// TIA Portal V20 export
FUNCTION "CollectAlarms" : Void   // FC66, LAD
TITLE = U1Em6_StackTable
// stored: Namespace Unit1.Em6, SetENOAutomatically false
   VAR_INPUT
      resetAlarms : Bool;
      disableAlarms : Bool;
   END_VAR
   VAR_OUTPUT
      commandsToUnit : "LUC_typeStateCommands";   // Feedback to the unit
   END_VAR
   VAR CONSTANT
      DelayTime : Time := T#300ms;
      NoDelayTime : Time;
      FALSE : Bool := FALSE;
      TRUE : Bool := TRUE;
   END_VAR
BEGIN

REGION Network 1: Reset Alarms
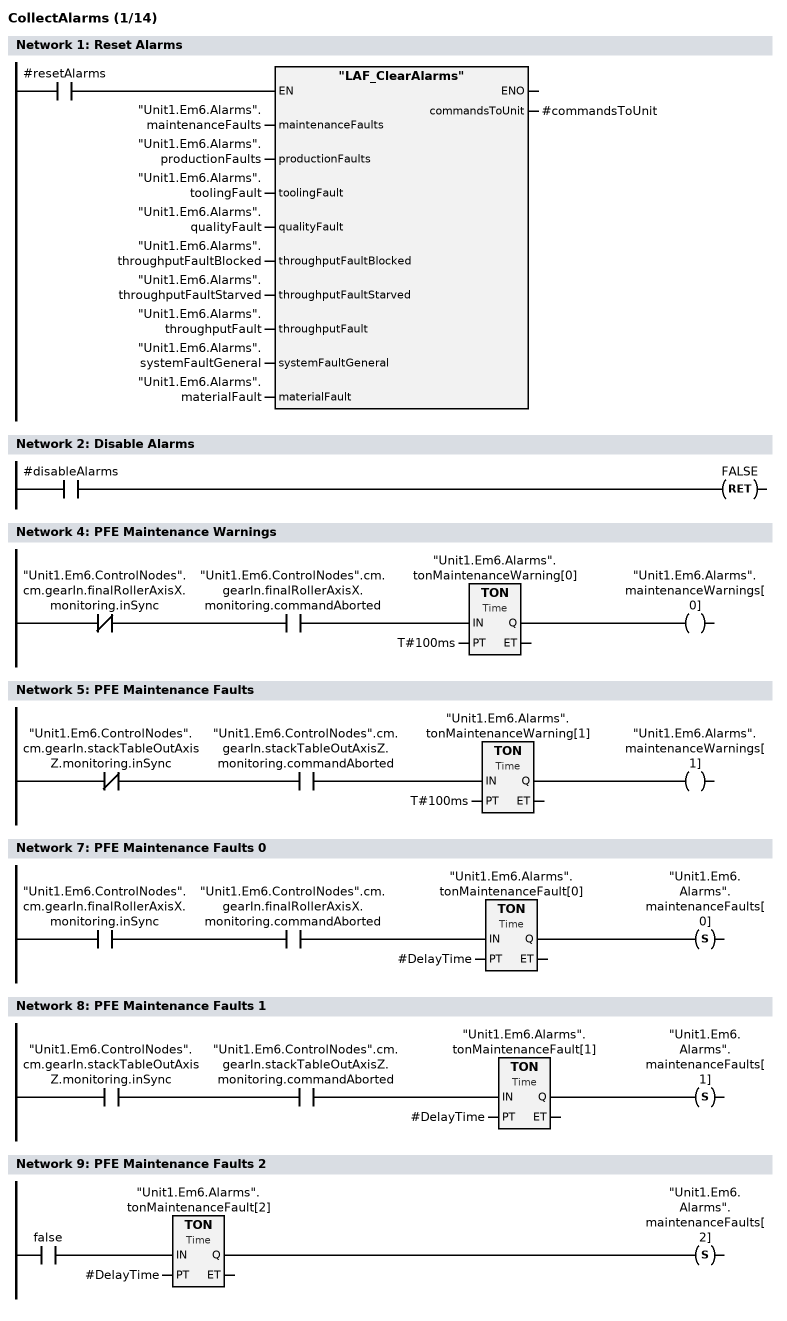
   RUNG wire#powerrail
      Contact( #resetAlarms )
      "LAF_ClearAlarms"(maintenanceFaults := "Unit1.Em6.Alarms".maintenanceFaults, productionFaults := "Unit1.Em6.Alarms".productionFaults, toolingFault := "Unit1.Em6.Alarms".toolingFault, qualityFault := "Unit1.Em6.Alarms".qualityFault, throughputFaultBlocked := "Unit1.Em6.Alarms".throughputFaultBlocked, throughputFaultStarved := "Unit1.Em6.Alarms".throughputFaultStarved, throughputFault := "Unit1.Em6.Alarms".throughputFault, systemFaultGeneral := "Unit1.Em6.Alarms".systemFaultGeneral, materialFault := "Unit1.Em6.Alarms".materialFault, commandsToUnit => #commandsToUnit)
   END_RUNG
   // the same network as SCL:
   IF #resetAlarms THEN
       "LAF_ClearAlarms"(maintenanceFaults := "Unit1.Em6.Alarms".maintenanceFaults,
                         productionFaults := "Unit1.Em6.Alarms".productionFaults,
                         toolingFault := "Unit1.Em6.Alarms".toolingFault,
                         qualityFault := "Unit1.Em6.Alarms".qualityFault,
                         throughputFaultBlocked := "Unit1.Em6.Alarms".throughputFaultBlocked,
                         throughputFaultStarved := "Unit1.Em6.Alarms".throughputFaultStarved,
                         throughputFault := "Unit1.Em6.Alarms".throughputFault,
                         systemFaultGeneral := "Unit1.Em6.Alarms".systemFaultGeneral,
                         materialFault := "Unit1.Em6.Alarms".materialFault,
                         commandsToUnit => #commandsToUnit);
   END_IF;
END_REGION

REGION Network 2: Disable Alarms
   RUNG wire#powerrail
      Contact( #disableAlarms )
      ReturnCoil( FALSE )
   END_RUNG
   // the same network as SCL:
   IF #disableAlarms THEN
       ENO := FALSE;
       RETURN;
   END_IF;
END_REGION

REGION Network 3: *************** Fault ************************
END_REGION

REGION Network 4: PFE Maintenance Warnings
   RUNG wire#powerrail
      I_Contact( "Unit1.Em6.ControlNodes".cm.gearIn.finalRollerAxisX.monitoring.inSync )
      Contact( "Unit1.Em6.ControlNodes".cm.gearIn.finalRollerAxisX.monitoring.commandAborted )
      { S7_Templates := "time_type := Time" } "Unit1.Em6.Alarms".tonMaintenanceWarning[0].TON(pt := T#100ms, et =>)
      Coil( "Unit1.Em6.Alarms".maintenanceWarnings[0] )
   END_RUNG
   // the same network as SCL:
   "Unit1.Em6.Alarms".tonMaintenanceWarning[0].TON(IN := NOT "Unit1.Em6.ControlNodes".cm.gearIn.finalRollerAxisX.monitoring.inSync AND "Unit1.Em6.ControlNodes".cm.gearIn.finalRollerAxisX.monitoring.commandAborted,
                           PT := T#100ms);
   "Unit1.Em6.Alarms".maintenanceWarnings[0] := "Unit1.Em6.Alarms".tonMaintenanceWarning[0].Q;
END_REGION

REGION Network 5: PFE Maintenance Faults
   RUNG wire#powerrail
      I_Contact( "Unit1.Em6.ControlNodes".cm.gearIn.stackTableOutAxisZ.monitoring.inSync )
      Contact( "Unit1.Em6.ControlNodes".cm.gearIn.stackTableOutAxisZ.monitoring.commandAborted )
      { S7_Templates := "time_type := Time" } "Unit1.Em6.Alarms".tonMaintenanceWarning[1].TON(pt := T#100ms, et =>)
      Coil( "Unit1.Em6.Alarms".maintenanceWarnings[1] )
   END_RUNG
   // the same network as SCL:
   "Unit1.Em6.Alarms".tonMaintenanceWarning[1].TON(IN := NOT "Unit1.Em6.ControlNodes".cm.gearIn.stackTableOutAxisZ.monitoring.inSync AND "Unit1.Em6.ControlNodes".cm.gearIn.stackTableOutAxisZ.monitoring.commandAborted,
                           PT := T#100ms);
   "Unit1.Em6.Alarms".maintenanceWarnings[1] := "Unit1.Em6.Alarms".tonMaintenanceWarning[1].Q;
END_REGION

REGION Network 7: PFE Maintenance Faults 0
   RUNG wire#powerrail
      Contact( "Unit1.Em6.ControlNodes".cm.gearIn.finalRollerAxisX.monitoring.inSync )
      Contact( "Unit1.Em6.ControlNodes".cm.gearIn.finalRollerAxisX.monitoring.commandAborted )
      { S7_Templates := "time_type := Time" } "Unit1.Em6.Alarms".tonMaintenanceFault[0].TON(pt := #DelayTime, et =>)
      S_Coil( "Unit1.Em6.Alarms".maintenanceFaults[0] )
   END_RUNG
   // the same network as SCL:
   "Unit1.Em6.Alarms".tonMaintenanceFault[0].TON(IN := "Unit1.Em6.ControlNodes".cm.gearIn.finalRollerAxisX.monitoring.inSync AND "Unit1.Em6.ControlNodes".cm.gearIn.finalRollerAxisX.monitoring.commandAborted,
                           PT := #DelayTime);
   IF "Unit1.Em6.Alarms".tonMaintenanceFault[0].Q THEN
       "Unit1.Em6.Alarms".maintenanceFaults[0] := TRUE;
   END_IF;
END_REGION

REGION Network 8: PFE Maintenance Faults 1
   RUNG wire#powerrail
      Contact( "Unit1.Em6.ControlNodes".cm.gearIn.stackTableOutAxisZ.monitoring.inSync )
      Contact( "Unit1.Em6.ControlNodes".cm.gearIn.stackTableOutAxisZ.monitoring.commandAborted )
      { S7_Templates := "time_type := Time" } "Unit1.Em6.Alarms".tonMaintenanceFault[1].TON(pt := #DelayTime, et =>)
      S_Coil( "Unit1.Em6.Alarms".maintenanceFaults[1] )
   END_RUNG
   // the same network as SCL:
   "Unit1.Em6.Alarms".tonMaintenanceFault[1].TON(IN := "Unit1.Em6.ControlNodes".cm.gearIn.stackTableOutAxisZ.monitoring.inSync AND "Unit1.Em6.ControlNodes".cm.gearIn.stackTableOutAxisZ.monitoring.commandAborted,
                           PT := #DelayTime);
   IF "Unit1.Em6.Alarms".tonMaintenanceFault[1].Q THEN
       "Unit1.Em6.Alarms".maintenanceFaults[1] := TRUE;
   END_IF;
END_REGION

REGION Network 9: PFE Maintenance Faults 2
   RUNG wire#powerrail
      Contact( false )
      { S7_Templates := "time_type := Time" } "Unit1.Em6.Alarms".tonMaintenanceFault[2].TON(pt := #DelayTime, et =>)
      S_Coil( "Unit1.Em6.Alarms".maintenanceFaults[2] )
   END_RUNG
   // the same network as SCL:
   "Unit1.Em6.Alarms".tonMaintenanceFault[2].TON(IN := false, PT := #DelayTime);
   IF "Unit1.Em6.Alarms".tonMaintenanceFault[2].Q THEN
       "Unit1.Em6.Alarms".maintenanceFaults[2] := TRUE;
   END_IF;
END_REGION

REGION Network 10: PFE Maintenance Faults 3
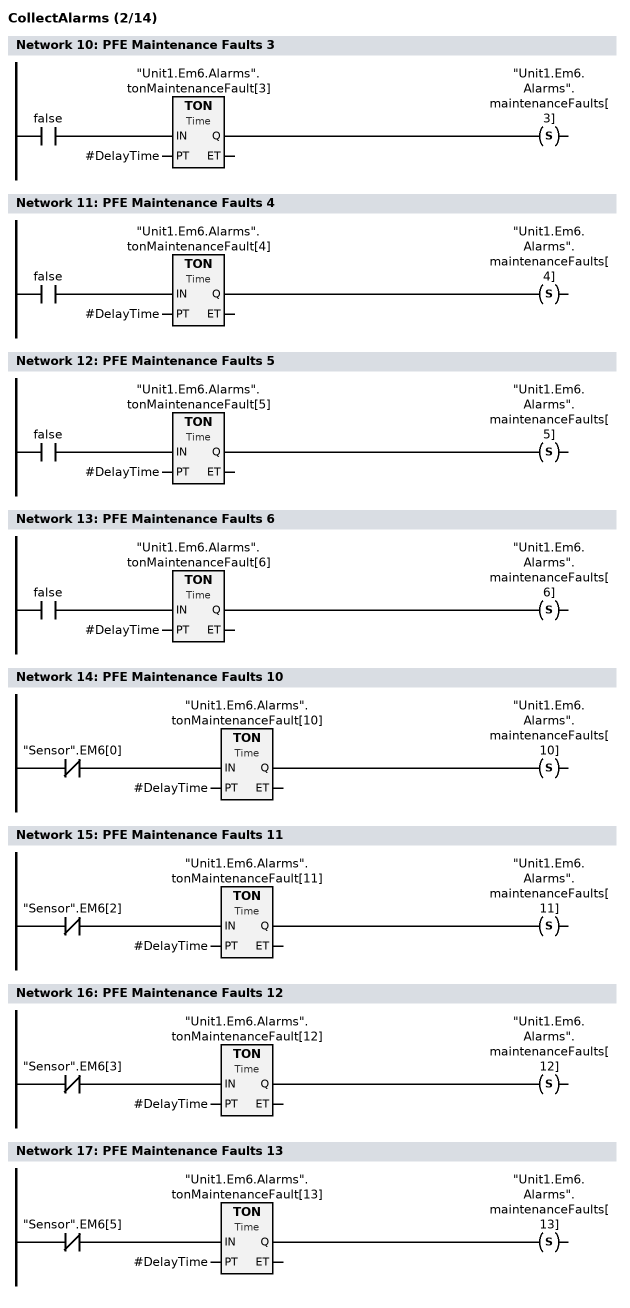
   RUNG wire#powerrail
      Contact( false )
      { S7_Templates := "time_type := Time" } "Unit1.Em6.Alarms".tonMaintenanceFault[3].TON(pt := #DelayTime, et =>)
      S_Coil( "Unit1.Em6.Alarms".maintenanceFaults[3] )
   END_RUNG
   // the same network as SCL:
   "Unit1.Em6.Alarms".tonMaintenanceFault[3].TON(IN := false, PT := #DelayTime);
   IF "Unit1.Em6.Alarms".tonMaintenanceFault[3].Q THEN
       "Unit1.Em6.Alarms".maintenanceFaults[3] := TRUE;
   END_IF;
END_REGION

REGION Network 11: PFE Maintenance Faults 4
   RUNG wire#powerrail
      Contact( false )
      { S7_Templates := "time_type := Time" } "Unit1.Em6.Alarms".tonMaintenanceFault[4].TON(pt := #DelayTime, et =>)
      S_Coil( "Unit1.Em6.Alarms".maintenanceFaults[4] )
   END_RUNG
   // the same network as SCL:
   "Unit1.Em6.Alarms".tonMaintenanceFault[4].TON(IN := false, PT := #DelayTime);
   IF "Unit1.Em6.Alarms".tonMaintenanceFault[4].Q THEN
       "Unit1.Em6.Alarms".maintenanceFaults[4] := TRUE;
   END_IF;
END_REGION

REGION Network 12: PFE Maintenance Faults 5
   RUNG wire#powerrail
      Contact( false )
      { S7_Templates := "time_type := Time" } "Unit1.Em6.Alarms".tonMaintenanceFault[5].TON(pt := #DelayTime, et =>)
      S_Coil( "Unit1.Em6.Alarms".maintenanceFaults[5] )
   END_RUNG
   // the same network as SCL:
   "Unit1.Em6.Alarms".tonMaintenanceFault[5].TON(IN := false, PT := #DelayTime);
   IF "Unit1.Em6.Alarms".tonMaintenanceFault[5].Q THEN
       "Unit1.Em6.Alarms".maintenanceFaults[5] := TRUE;
   END_IF;
END_REGION

REGION Network 13: PFE Maintenance Faults 6
   RUNG wire#powerrail
      Contact( false )
      { S7_Templates := "time_type := Time" } "Unit1.Em6.Alarms".tonMaintenanceFault[6].TON(pt := #DelayTime, et =>)
      S_Coil( "Unit1.Em6.Alarms".maintenanceFaults[6] )
   END_RUNG
   // the same network as SCL:
   "Unit1.Em6.Alarms".tonMaintenanceFault[6].TON(IN := false, PT := #DelayTime);
   IF "Unit1.Em6.Alarms".tonMaintenanceFault[6].Q THEN
       "Unit1.Em6.Alarms".maintenanceFaults[6] := TRUE;
   END_IF;
END_REGION

REGION Network 14: PFE Maintenance Faults 10
   RUNG wire#powerrail
      I_Contact( "Sensor".EM6[0] )
      { S7_Templates := "time_type := Time" } "Unit1.Em6.Alarms".tonMaintenanceFault[10].TON(pt := #DelayTime, et =>)
      S_Coil( "Unit1.Em6.Alarms".maintenanceFaults[10] )
   END_RUNG
   // the same network as SCL:
   "Unit1.Em6.Alarms".tonMaintenanceFault[10].TON(IN := NOT "Sensor".EM6[0], PT := #DelayTime);
   IF "Unit1.Em6.Alarms".tonMaintenanceFault[10].Q THEN
       "Unit1.Em6.Alarms".maintenanceFaults[10] := TRUE;
   END_IF;
END_REGION

REGION Network 15: PFE Maintenance Faults 11
   RUNG wire#powerrail
      I_Contact( "Sensor".EM6[2] )
      { S7_Templates := "time_type := Time" } "Unit1.Em6.Alarms".tonMaintenanceFault[11].TON(pt := #DelayTime, et =>)
      S_Coil( "Unit1.Em6.Alarms".maintenanceFaults[11] )
   END_RUNG
   // the same network as SCL:
   "Unit1.Em6.Alarms".tonMaintenanceFault[11].TON(IN := NOT "Sensor".EM6[2], PT := #DelayTime);
   IF "Unit1.Em6.Alarms".tonMaintenanceFault[11].Q THEN
       "Unit1.Em6.Alarms".maintenanceFaults[11] := TRUE;
   END_IF;
END_REGION

REGION Network 16: PFE Maintenance Faults 12
   RUNG wire#powerrail
      I_Contact( "Sensor".EM6[3] )
      { S7_Templates := "time_type := Time" } "Unit1.Em6.Alarms".tonMaintenanceFault[12].TON(pt := #DelayTime, et =>)
      S_Coil( "Unit1.Em6.Alarms".maintenanceFaults[12] )
   END_RUNG
   // the same network as SCL:
   "Unit1.Em6.Alarms".tonMaintenanceFault[12].TON(IN := NOT "Sensor".EM6[3], PT := #DelayTime);
   IF "Unit1.Em6.Alarms".tonMaintenanceFault[12].Q THEN
       "Unit1.Em6.Alarms".maintenanceFaults[12] := TRUE;
   END_IF;
END_REGION

REGION Network 17: PFE Maintenance Faults 13
   RUNG wire#powerrail
      I_Contact( "Sensor".EM6[5] )
      { S7_Templates := "time_type := Time" } "Unit1.Em6.Alarms".tonMaintenanceFault[13].TON(pt := #DelayTime, et =>)
      S_Coil( "Unit1.Em6.Alarms".maintenanceFaults[13] )
   END_RUNG
   // the same network as SCL:
   "Unit1.Em6.Alarms".tonMaintenanceFault[13].TON(IN := NOT "Sensor".EM6[5], PT := #DelayTime);
   IF "Unit1.Em6.Alarms".tonMaintenanceFault[13].Q THEN
       "Unit1.Em6.Alarms".maintenanceFaults[13] := TRUE;
   END_IF;
END_REGION

REGION Network 18: PFE Maintenance Faults 14
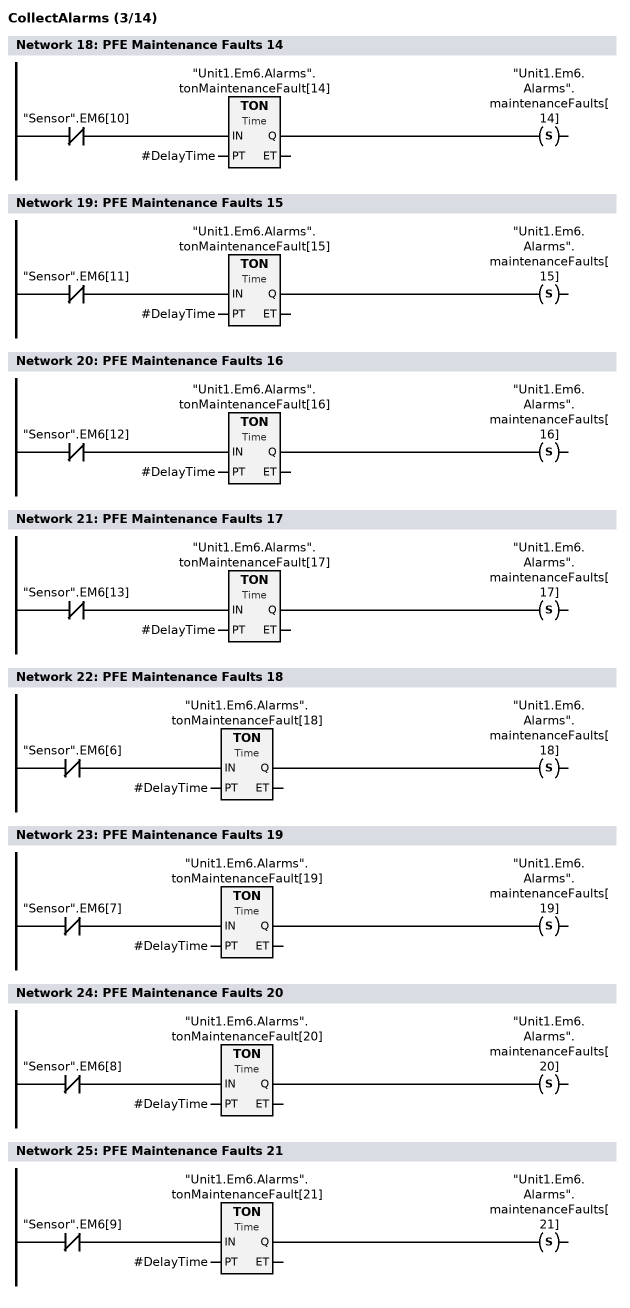
   RUNG wire#powerrail
      I_Contact( "Sensor".EM6[10] )
      { S7_Templates := "time_type := Time" } "Unit1.Em6.Alarms".tonMaintenanceFault[14].TON(pt := #DelayTime, et =>)
      S_Coil( "Unit1.Em6.Alarms".maintenanceFaults[14] )
   END_RUNG
   // the same network as SCL:
   "Unit1.Em6.Alarms".tonMaintenanceFault[14].TON(IN := NOT "Sensor".EM6[10], PT := #DelayTime);
   IF "Unit1.Em6.Alarms".tonMaintenanceFault[14].Q THEN
       "Unit1.Em6.Alarms".maintenanceFaults[14] := TRUE;
   END_IF;
END_REGION

REGION Network 19: PFE Maintenance Faults 15
   RUNG wire#powerrail
      I_Contact( "Sensor".EM6[11] )
      { S7_Templates := "time_type := Time" } "Unit1.Em6.Alarms".tonMaintenanceFault[15].TON(pt := #DelayTime, et =>)
      S_Coil( "Unit1.Em6.Alarms".maintenanceFaults[15] )
   END_RUNG
   // the same network as SCL:
   "Unit1.Em6.Alarms".tonMaintenanceFault[15].TON(IN := NOT "Sensor".EM6[11], PT := #DelayTime);
   IF "Unit1.Em6.Alarms".tonMaintenanceFault[15].Q THEN
       "Unit1.Em6.Alarms".maintenanceFaults[15] := TRUE;
   END_IF;
END_REGION

REGION Network 20: PFE Maintenance Faults 16
   RUNG wire#powerrail
      I_Contact( "Sensor".EM6[12] )
      { S7_Templates := "time_type := Time" } "Unit1.Em6.Alarms".tonMaintenanceFault[16].TON(pt := #DelayTime, et =>)
      S_Coil( "Unit1.Em6.Alarms".maintenanceFaults[16] )
   END_RUNG
   // the same network as SCL:
   "Unit1.Em6.Alarms".tonMaintenanceFault[16].TON(IN := NOT "Sensor".EM6[12], PT := #DelayTime);
   IF "Unit1.Em6.Alarms".tonMaintenanceFault[16].Q THEN
       "Unit1.Em6.Alarms".maintenanceFaults[16] := TRUE;
   END_IF;
END_REGION

REGION Network 21: PFE Maintenance Faults 17
   RUNG wire#powerrail
      I_Contact( "Sensor".EM6[13] )
      { S7_Templates := "time_type := Time" } "Unit1.Em6.Alarms".tonMaintenanceFault[17].TON(pt := #DelayTime, et =>)
      S_Coil( "Unit1.Em6.Alarms".maintenanceFaults[17] )
   END_RUNG
   // the same network as SCL:
   "Unit1.Em6.Alarms".tonMaintenanceFault[17].TON(IN := NOT "Sensor".EM6[13], PT := #DelayTime);
   IF "Unit1.Em6.Alarms".tonMaintenanceFault[17].Q THEN
       "Unit1.Em6.Alarms".maintenanceFaults[17] := TRUE;
   END_IF;
END_REGION

REGION Network 22: PFE Maintenance Faults 18
   RUNG wire#powerrail
      I_Contact( "Sensor".EM6[6] )
      { S7_Templates := "time_type := Time" } "Unit1.Em6.Alarms".tonMaintenanceFault[18].TON(pt := #DelayTime, et =>)
      S_Coil( "Unit1.Em6.Alarms".maintenanceFaults[18] )
   END_RUNG
   // the same network as SCL:
   "Unit1.Em6.Alarms".tonMaintenanceFault[18].TON(IN := NOT "Sensor".EM6[6], PT := #DelayTime);
   IF "Unit1.Em6.Alarms".tonMaintenanceFault[18].Q THEN
       "Unit1.Em6.Alarms".maintenanceFaults[18] := TRUE;
   END_IF;
END_REGION

REGION Network 23: PFE Maintenance Faults 19
   RUNG wire#powerrail
      I_Contact( "Sensor".EM6[7] )
      { S7_Templates := "time_type := Time" } "Unit1.Em6.Alarms".tonMaintenanceFault[19].TON(pt := #DelayTime, et =>)
      S_Coil( "Unit1.Em6.Alarms".maintenanceFaults[19] )
   END_RUNG
   // the same network as SCL:
   "Unit1.Em6.Alarms".tonMaintenanceFault[19].TON(IN := NOT "Sensor".EM6[7], PT := #DelayTime);
   IF "Unit1.Em6.Alarms".tonMaintenanceFault[19].Q THEN
       "Unit1.Em6.Alarms".maintenanceFaults[19] := TRUE;
   END_IF;
END_REGION

REGION Network 24: PFE Maintenance Faults 20
   RUNG wire#powerrail
      I_Contact( "Sensor".EM6[8] )
      { S7_Templates := "time_type := Time" } "Unit1.Em6.Alarms".tonMaintenanceFault[20].TON(pt := #DelayTime, et =>)
      S_Coil( "Unit1.Em6.Alarms".maintenanceFaults[20] )
   END_RUNG
   // the same network as SCL:
   "Unit1.Em6.Alarms".tonMaintenanceFault[20].TON(IN := NOT "Sensor".EM6[8], PT := #DelayTime);
   IF "Unit1.Em6.Alarms".tonMaintenanceFault[20].Q THEN
       "Unit1.Em6.Alarms".maintenanceFaults[20] := TRUE;
   END_IF;
END_REGION

REGION Network 25: PFE Maintenance Faults 21
   RUNG wire#powerrail
      I_Contact( "Sensor".EM6[9] )
      { S7_Templates := "time_type := Time" } "Unit1.Em6.Alarms".tonMaintenanceFault[21].TON(pt := #DelayTime, et =>)
      S_Coil( "Unit1.Em6.Alarms".maintenanceFaults[21] )
   END_RUNG
   // the same network as SCL:
   "Unit1.Em6.Alarms".tonMaintenanceFault[21].TON(IN := NOT "Sensor".EM6[9], PT := #DelayTime);
   IF "Unit1.Em6.Alarms".tonMaintenanceFault[21].Q THEN
       "Unit1.Em6.Alarms".maintenanceFaults[21] := TRUE;
   END_IF;
END_REGION

REGION Network 26: PFE Maintenance Faults 22
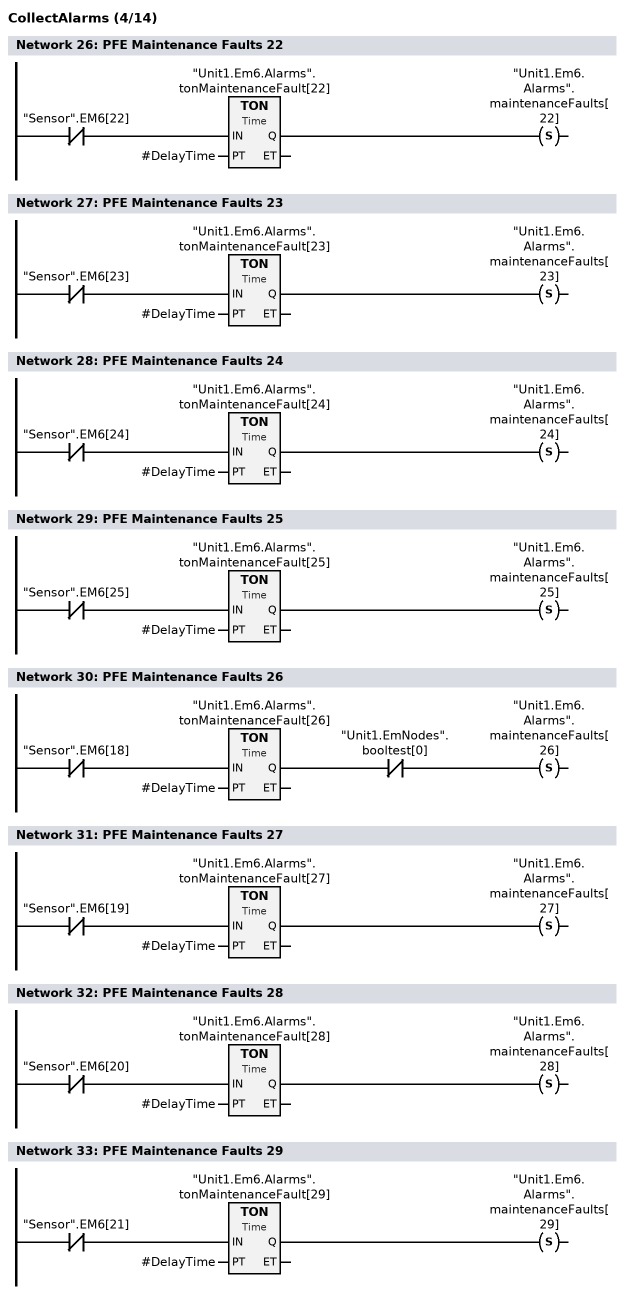
   RUNG wire#powerrail
      I_Contact( "Sensor".EM6[22] )
      { S7_Templates := "time_type := Time" } "Unit1.Em6.Alarms".tonMaintenanceFault[22].TON(pt := #DelayTime, et =>)
      S_Coil( "Unit1.Em6.Alarms".maintenanceFaults[22] )
   END_RUNG
   // the same network as SCL:
   "Unit1.Em6.Alarms".tonMaintenanceFault[22].TON(IN := NOT "Sensor".EM6[22], PT := #DelayTime);
   IF "Unit1.Em6.Alarms".tonMaintenanceFault[22].Q THEN
       "Unit1.Em6.Alarms".maintenanceFaults[22] := TRUE;
   END_IF;
END_REGION

REGION Network 27: PFE Maintenance Faults 23
   RUNG wire#powerrail
      I_Contact( "Sensor".EM6[23] )
      { S7_Templates := "time_type := Time" } "Unit1.Em6.Alarms".tonMaintenanceFault[23].TON(pt := #DelayTime, et =>)
      S_Coil( "Unit1.Em6.Alarms".maintenanceFaults[23] )
   END_RUNG
   // the same network as SCL:
   "Unit1.Em6.Alarms".tonMaintenanceFault[23].TON(IN := NOT "Sensor".EM6[23], PT := #DelayTime);
   IF "Unit1.Em6.Alarms".tonMaintenanceFault[23].Q THEN
       "Unit1.Em6.Alarms".maintenanceFaults[23] := TRUE;
   END_IF;
END_REGION

REGION Network 28: PFE Maintenance Faults 24
   RUNG wire#powerrail
      I_Contact( "Sensor".EM6[24] )
      { S7_Templates := "time_type := Time" } "Unit1.Em6.Alarms".tonMaintenanceFault[24].TON(pt := #DelayTime, et =>)
      S_Coil( "Unit1.Em6.Alarms".maintenanceFaults[24] )
   END_RUNG
   // the same network as SCL:
   "Unit1.Em6.Alarms".tonMaintenanceFault[24].TON(IN := NOT "Sensor".EM6[24], PT := #DelayTime);
   IF "Unit1.Em6.Alarms".tonMaintenanceFault[24].Q THEN
       "Unit1.Em6.Alarms".maintenanceFaults[24] := TRUE;
   END_IF;
END_REGION

REGION Network 29: PFE Maintenance Faults 25
   RUNG wire#powerrail
      I_Contact( "Sensor".EM6[25] )
      { S7_Templates := "time_type := Time" } "Unit1.Em6.Alarms".tonMaintenanceFault[25].TON(pt := #DelayTime, et =>)
      S_Coil( "Unit1.Em6.Alarms".maintenanceFaults[25] )
   END_RUNG
   // the same network as SCL:
   "Unit1.Em6.Alarms".tonMaintenanceFault[25].TON(IN := NOT "Sensor".EM6[25], PT := #DelayTime);
   IF "Unit1.Em6.Alarms".tonMaintenanceFault[25].Q THEN
       "Unit1.Em6.Alarms".maintenanceFaults[25] := TRUE;
   END_IF;
END_REGION

REGION Network 30: PFE Maintenance Faults 26
   RUNG wire#powerrail
      I_Contact( "Sensor".EM6[18] )
      { S7_Templates := "time_type := Time" } "Unit1.Em6.Alarms".tonMaintenanceFault[26].TON(pt := #DelayTime, et =>)
      I_Contact( "Unit1.EmNodes".booltest[0] )
      S_Coil( "Unit1.Em6.Alarms".maintenanceFaults[26] )
   END_RUNG
   // the same network as SCL:
   "Unit1.Em6.Alarms".tonMaintenanceFault[26].TON(IN := NOT "Sensor".EM6[18], PT := #DelayTime);
   IF "Unit1.Em6.Alarms".tonMaintenanceFault[26].Q AND NOT "Unit1.EmNodes".booltest[0] THEN
       "Unit1.Em6.Alarms".maintenanceFaults[26] := TRUE;
   END_IF;
END_REGION

REGION Network 31: PFE Maintenance Faults 27
   RUNG wire#powerrail
      I_Contact( "Sensor".EM6[19] )
      { S7_Templates := "time_type := Time" } "Unit1.Em6.Alarms".tonMaintenanceFault[27].TON(pt := #DelayTime, et =>)
      S_Coil( "Unit1.Em6.Alarms".maintenanceFaults[27] )
   END_RUNG
   // the same network as SCL:
   "Unit1.Em6.Alarms".tonMaintenanceFault[27].TON(IN := NOT "Sensor".EM6[19], PT := #DelayTime);
   IF "Unit1.Em6.Alarms".tonMaintenanceFault[27].Q THEN
       "Unit1.Em6.Alarms".maintenanceFaults[27] := TRUE;
   END_IF;
END_REGION

REGION Network 32: PFE Maintenance Faults 28
   RUNG wire#powerrail
      I_Contact( "Sensor".EM6[20] )
      { S7_Templates := "time_type := Time" } "Unit1.Em6.Alarms".tonMaintenanceFault[28].TON(pt := #DelayTime, et =>)
      S_Coil( "Unit1.Em6.Alarms".maintenanceFaults[28] )
   END_RUNG
   // the same network as SCL:
   "Unit1.Em6.Alarms".tonMaintenanceFault[28].TON(IN := NOT "Sensor".EM6[20], PT := #DelayTime);
   IF "Unit1.Em6.Alarms".tonMaintenanceFault[28].Q THEN
       "Unit1.Em6.Alarms".maintenanceFaults[28] := TRUE;
   END_IF;
END_REGION

REGION Network 33: PFE Maintenance Faults 29
   RUNG wire#powerrail
      I_Contact( "Sensor".EM6[21] )
      { S7_Templates := "time_type := Time" } "Unit1.Em6.Alarms".tonMaintenanceFault[29].TON(pt := #DelayTime, et =>)
      S_Coil( "Unit1.Em6.Alarms".maintenanceFaults[29] )
   END_RUNG
   // the same network as SCL:
   "Unit1.Em6.Alarms".tonMaintenanceFault[29].TON(IN := NOT "Sensor".EM6[21], PT := #DelayTime);
   IF "Unit1.Em6.Alarms".tonMaintenanceFault[29].Q THEN
       "Unit1.Em6.Alarms".maintenanceFaults[29] := TRUE;
   END_IF;
END_REGION

REGION Network 34: PFE Maintenance Faults 30
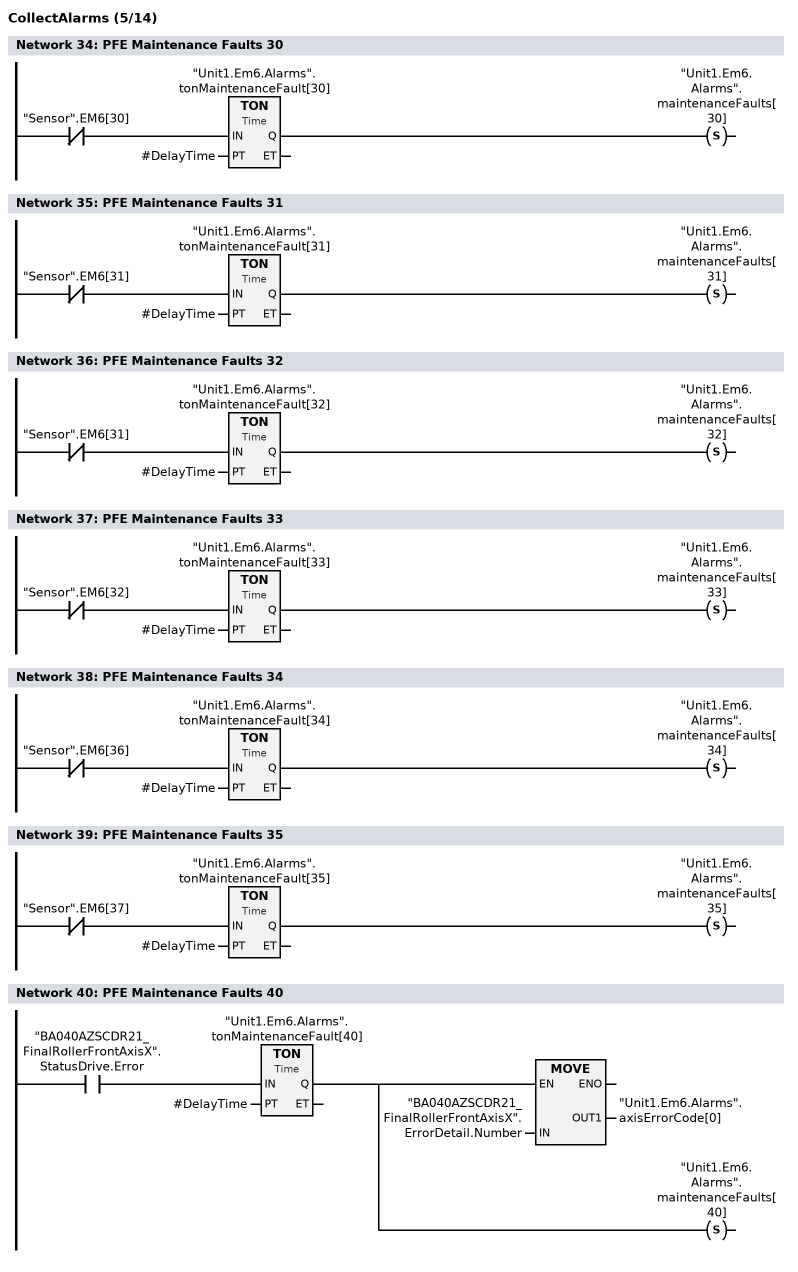
   RUNG wire#powerrail
      I_Contact( "Sensor".EM6[30] )
      { S7_Templates := "time_type := Time" } "Unit1.Em6.Alarms".tonMaintenanceFault[30].TON(pt := #DelayTime, et =>)
      S_Coil( "Unit1.Em6.Alarms".maintenanceFaults[30] )
   END_RUNG
   // the same network as SCL:
   "Unit1.Em6.Alarms".tonMaintenanceFault[30].TON(IN := NOT "Sensor".EM6[30], PT := #DelayTime);
   IF "Unit1.Em6.Alarms".tonMaintenanceFault[30].Q THEN
       "Unit1.Em6.Alarms".maintenanceFaults[30] := TRUE;
   END_IF;
END_REGION

REGION Network 35: PFE Maintenance Faults 31
   RUNG wire#powerrail
      I_Contact( "Sensor".EM6[31] )
      { S7_Templates := "time_type := Time" } "Unit1.Em6.Alarms".tonMaintenanceFault[31].TON(pt := #DelayTime, et =>)
      S_Coil( "Unit1.Em6.Alarms".maintenanceFaults[31] )
   END_RUNG
   // the same network as SCL:
   "Unit1.Em6.Alarms".tonMaintenanceFault[31].TON(IN := NOT "Sensor".EM6[31], PT := #DelayTime);
   IF "Unit1.Em6.Alarms".tonMaintenanceFault[31].Q THEN
       "Unit1.Em6.Alarms".maintenanceFaults[31] := TRUE;
   END_IF;
END_REGION

REGION Network 36: PFE Maintenance Faults 32
   RUNG wire#powerrail
      I_Contact( "Sensor".EM6[31] )
      { S7_Templates := "time_type := Time" } "Unit1.Em6.Alarms".tonMaintenanceFault[32].TON(pt := #DelayTime, et =>)
      S_Coil( "Unit1.Em6.Alarms".maintenanceFaults[32] )
   END_RUNG
   // the same network as SCL:
   "Unit1.Em6.Alarms".tonMaintenanceFault[32].TON(IN := NOT "Sensor".EM6[31], PT := #DelayTime);
   IF "Unit1.Em6.Alarms".tonMaintenanceFault[32].Q THEN
       "Unit1.Em6.Alarms".maintenanceFaults[32] := TRUE;
   END_IF;
END_REGION

REGION Network 37: PFE Maintenance Faults 33
   RUNG wire#powerrail
      I_Contact( "Sensor".EM6[32] )
      { S7_Templates := "time_type := Time" } "Unit1.Em6.Alarms".tonMaintenanceFault[33].TON(pt := #DelayTime, et =>)
      S_Coil( "Unit1.Em6.Alarms".maintenanceFaults[33] )
   END_RUNG
   // the same network as SCL:
   "Unit1.Em6.Alarms".tonMaintenanceFault[33].TON(IN := NOT "Sensor".EM6[32], PT := #DelayTime);
   IF "Unit1.Em6.Alarms".tonMaintenanceFault[33].Q THEN
       "Unit1.Em6.Alarms".maintenanceFaults[33] := TRUE;
   END_IF;
END_REGION

REGION Network 38: PFE Maintenance Faults 34
   RUNG wire#powerrail
      I_Contact( "Sensor".EM6[36] )
      { S7_Templates := "time_type := Time" } "Unit1.Em6.Alarms".tonMaintenanceFault[34].TON(pt := #DelayTime, et =>)
      S_Coil( "Unit1.Em6.Alarms".maintenanceFaults[34] )
   END_RUNG
   // the same network as SCL:
   "Unit1.Em6.Alarms".tonMaintenanceFault[34].TON(IN := NOT "Sensor".EM6[36], PT := #DelayTime);
   IF "Unit1.Em6.Alarms".tonMaintenanceFault[34].Q THEN
       "Unit1.Em6.Alarms".maintenanceFaults[34] := TRUE;
   END_IF;
END_REGION

REGION Network 39: PFE Maintenance Faults 35
   RUNG wire#powerrail
      I_Contact( "Sensor".EM6[37] )
      { S7_Templates := "time_type := Time" } "Unit1.Em6.Alarms".tonMaintenanceFault[35].TON(pt := #DelayTime, et =>)
      S_Coil( "Unit1.Em6.Alarms".maintenanceFaults[35] )
   END_RUNG
   // the same network as SCL:
   "Unit1.Em6.Alarms".tonMaintenanceFault[35].TON(IN := NOT "Sensor".EM6[37], PT := #DelayTime);
   IF "Unit1.Em6.Alarms".tonMaintenanceFault[35].Q THEN
       "Unit1.Em6.Alarms".maintenanceFaults[35] := TRUE;
   END_IF;
END_REGION

REGION Network 40: PFE Maintenance Faults 40
   RUNG wire#powerrail
      Contact( "BA040AZSCDR21_FinalRollerFrontAxisX".StatusDrive.Error )
      { S7_Templates := "time_type := Time" } "Unit1.Em6.Alarms".tonMaintenanceFault[40].TON(pt := #DelayTime, et =>)
      wire#w1
      Move(in := "BA040AZSCDR21_FinalRollerFrontAxisX".ErrorDetail.Number, out1 => "Unit1.Em6.Alarms".axisErrorCode[0])
   END_RUNG
   RUNG wire#w1
      S_Coil( "Unit1.Em6.Alarms".maintenanceFaults[40] )
   END_RUNG
   // the same network as SCL:
   "Unit1.Em6.Alarms".tonMaintenanceFault[40].TON(IN := "BA040AZSCDR21_FinalRollerFrontAxisX".StatusDrive.Error,
                           PT := #DelayTime);
   IF "Unit1.Em6.Alarms".tonMaintenanceFault[40].Q THEN
       "Unit1.Em6.Alarms".axisErrorCode[0] := "BA040AZSCDR21_FinalRollerFrontAxisX".ErrorDetail.Number;
       "Unit1.Em6.Alarms".maintenanceFaults[40] := TRUE;
   END_IF;
END_REGION

REGION Network 41: PFE Maintenance Faults 41
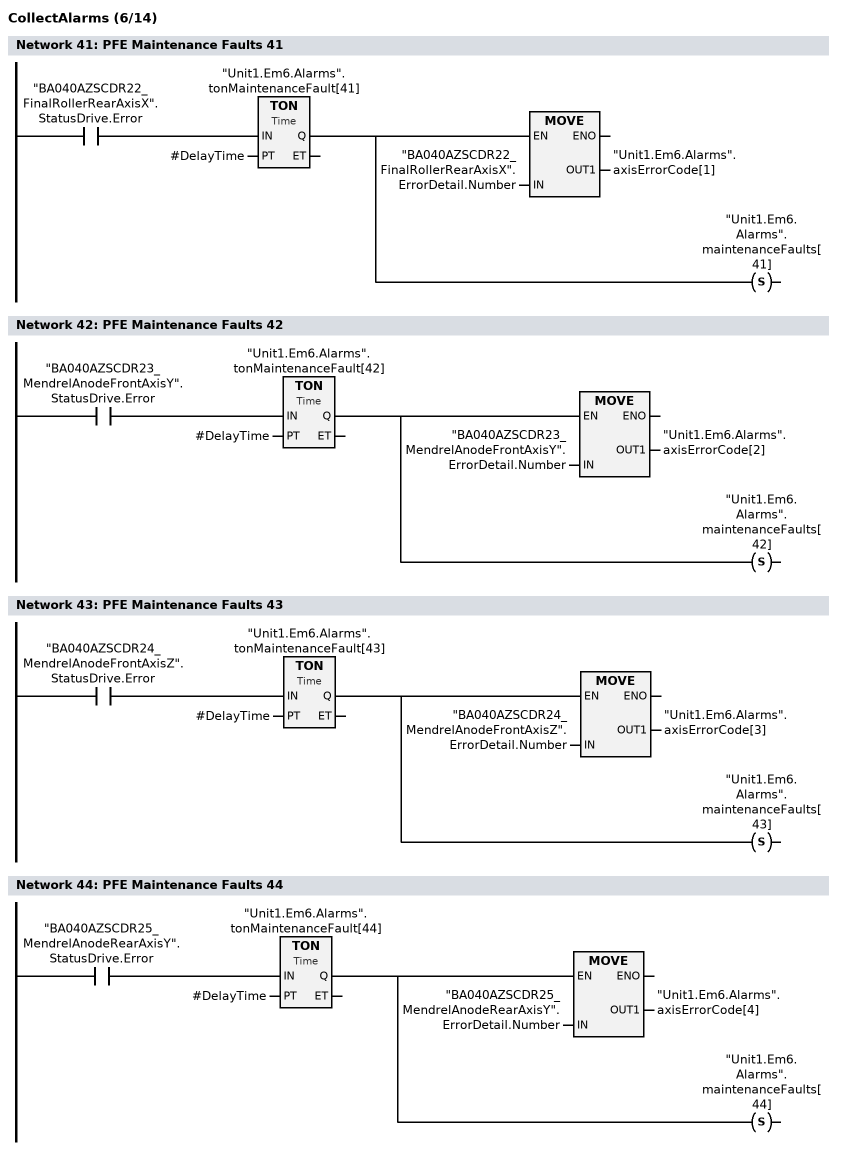
   RUNG wire#powerrail
      Contact( "BA040AZSCDR22_FinalRollerRearAxisX".StatusDrive.Error )
      { S7_Templates := "time_type := Time" } "Unit1.Em6.Alarms".tonMaintenanceFault[41].TON(pt := #DelayTime, et =>)
      wire#w1
      Move(in := "BA040AZSCDR22_FinalRollerRearAxisX".ErrorDetail.Number, out1 => "Unit1.Em6.Alarms".axisErrorCode[1])
   END_RUNG
   RUNG wire#w1
      S_Coil( "Unit1.Em6.Alarms".maintenanceFaults[41] )
   END_RUNG
   // the same network as SCL:
   "Unit1.Em6.Alarms".tonMaintenanceFault[41].TON(IN := "BA040AZSCDR22_FinalRollerRearAxisX".StatusDrive.Error,
                           PT := #DelayTime);
   IF "Unit1.Em6.Alarms".tonMaintenanceFault[41].Q THEN
       "Unit1.Em6.Alarms".axisErrorCode[1] := "BA040AZSCDR22_FinalRollerRearAxisX".ErrorDetail.Number;
       "Unit1.Em6.Alarms".maintenanceFaults[41] := TRUE;
   END_IF;
END_REGION

REGION Network 42: PFE Maintenance Faults 42
   RUNG wire#powerrail
      Contact( "BA040AZSCDR23_MendrelAnodeFrontAxisY".StatusDrive.Error )
      { S7_Templates := "time_type := Time" } "Unit1.Em6.Alarms".tonMaintenanceFault[42].TON(pt := #DelayTime, et =>)
      wire#w1
      Move(in := "BA040AZSCDR23_MendrelAnodeFrontAxisY".ErrorDetail.Number, out1 => "Unit1.Em6.Alarms".axisErrorCode[2])
   END_RUNG
   RUNG wire#w1
      S_Coil( "Unit1.Em6.Alarms".maintenanceFaults[42] )
   END_RUNG
   // the same network as SCL:
   "Unit1.Em6.Alarms".tonMaintenanceFault[42].TON(IN := "BA040AZSCDR23_MendrelAnodeFrontAxisY".StatusDrive.Error,
                           PT := #DelayTime);
   IF "Unit1.Em6.Alarms".tonMaintenanceFault[42].Q THEN
       "Unit1.Em6.Alarms".axisErrorCode[2] := "BA040AZSCDR23_MendrelAnodeFrontAxisY".ErrorDetail.Number;
       "Unit1.Em6.Alarms".maintenanceFaults[42] := TRUE;
   END_IF;
END_REGION

REGION Network 43: PFE Maintenance Faults 43
   RUNG wire#powerrail
      Contact( "BA040AZSCDR24_MendrelAnodeFrontAxisZ".StatusDrive.Error )
      { S7_Templates := "time_type := Time" } "Unit1.Em6.Alarms".tonMaintenanceFault[43].TON(pt := #DelayTime, et =>)
      wire#w1
      Move(in := "BA040AZSCDR24_MendrelAnodeFrontAxisZ".ErrorDetail.Number, out1 => "Unit1.Em6.Alarms".axisErrorCode[3])
   END_RUNG
   RUNG wire#w1
      S_Coil( "Unit1.Em6.Alarms".maintenanceFaults[43] )
   END_RUNG
   // the same network as SCL:
   "Unit1.Em6.Alarms".tonMaintenanceFault[43].TON(IN := "BA040AZSCDR24_MendrelAnodeFrontAxisZ".StatusDrive.Error,
                           PT := #DelayTime);
   IF "Unit1.Em6.Alarms".tonMaintenanceFault[43].Q THEN
       "Unit1.Em6.Alarms".axisErrorCode[3] := "BA040AZSCDR24_MendrelAnodeFrontAxisZ".ErrorDetail.Number;
       "Unit1.Em6.Alarms".maintenanceFaults[43] := TRUE;
   END_IF;
END_REGION

REGION Network 44: PFE Maintenance Faults 44
   RUNG wire#powerrail
      Contact( "BA040AZSCDR25_MendrelAnodeRearAxisY".StatusDrive.Error )
      { S7_Templates := "time_type := Time" } "Unit1.Em6.Alarms".tonMaintenanceFault[44].TON(pt := #DelayTime, et =>)
      wire#w1
      Move(in := "BA040AZSCDR25_MendrelAnodeRearAxisY".ErrorDetail.Number, out1 => "Unit1.Em6.Alarms".axisErrorCode[4])
   END_RUNG
   RUNG wire#w1
      S_Coil( "Unit1.Em6.Alarms".maintenanceFaults[44] )
   END_RUNG
   // the same network as SCL:
   "Unit1.Em6.Alarms".tonMaintenanceFault[44].TON(IN := "BA040AZSCDR25_MendrelAnodeRearAxisY".StatusDrive.Error,
                           PT := #DelayTime);
   IF "Unit1.Em6.Alarms".tonMaintenanceFault[44].Q THEN
       "Unit1.Em6.Alarms".axisErrorCode[4] := "BA040AZSCDR25_MendrelAnodeRearAxisY".ErrorDetail.Number;
       "Unit1.Em6.Alarms".maintenanceFaults[44] := TRUE;
   END_IF;
END_REGION

REGION Network 45: PFE Maintenance Faults 45
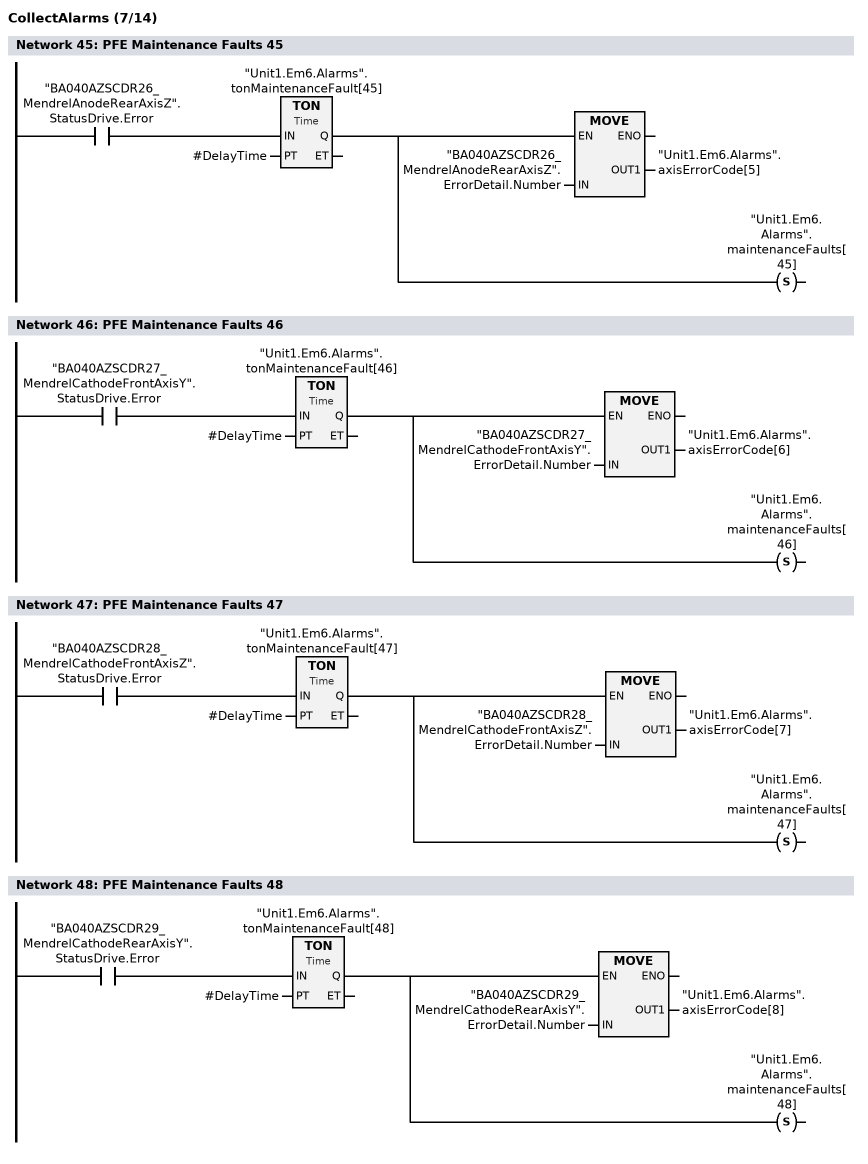
   RUNG wire#powerrail
      Contact( "BA040AZSCDR26_MendrelAnodeRearAxisZ".StatusDrive.Error )
      { S7_Templates := "time_type := Time" } "Unit1.Em6.Alarms".tonMaintenanceFault[45].TON(pt := #DelayTime, et =>)
      wire#w1
      Move(in := "BA040AZSCDR26_MendrelAnodeRearAxisZ".ErrorDetail.Number, out1 => "Unit1.Em6.Alarms".axisErrorCode[5])
   END_RUNG
   RUNG wire#w1
      S_Coil( "Unit1.Em6.Alarms".maintenanceFaults[45] )
   END_RUNG
   // the same network as SCL:
   "Unit1.Em6.Alarms".tonMaintenanceFault[45].TON(IN := "BA040AZSCDR26_MendrelAnodeRearAxisZ".StatusDrive.Error,
                           PT := #DelayTime);
   IF "Unit1.Em6.Alarms".tonMaintenanceFault[45].Q THEN
       "Unit1.Em6.Alarms".axisErrorCode[5] := "BA040AZSCDR26_MendrelAnodeRearAxisZ".ErrorDetail.Number;
       "Unit1.Em6.Alarms".maintenanceFaults[45] := TRUE;
   END_IF;
END_REGION

REGION Network 46: PFE Maintenance Faults 46
   RUNG wire#powerrail
      Contact( "BA040AZSCDR27_MendrelCathodeFrontAxisY".StatusDrive.Error )
      { S7_Templates := "time_type := Time" } "Unit1.Em6.Alarms".tonMaintenanceFault[46].TON(pt := #DelayTime, et =>)
      wire#w1
      Move(in := "BA040AZSCDR27_MendrelCathodeFrontAxisY".ErrorDetail.Number, out1 => "Unit1.Em6.Alarms".axisErrorCode[6])
   END_RUNG
   RUNG wire#w1
      S_Coil( "Unit1.Em6.Alarms".maintenanceFaults[46] )
   END_RUNG
   // the same network as SCL:
   "Unit1.Em6.Alarms".tonMaintenanceFault[46].TON(IN := "BA040AZSCDR27_MendrelCathodeFrontAxisY".StatusDrive.Error,
                           PT := #DelayTime);
   IF "Unit1.Em6.Alarms".tonMaintenanceFault[46].Q THEN
       "Unit1.Em6.Alarms".axisErrorCode[6] := "BA040AZSCDR27_MendrelCathodeFrontAxisY".ErrorDetail.Number;
       "Unit1.Em6.Alarms".maintenanceFaults[46] := TRUE;
   END_IF;
END_REGION

REGION Network 47: PFE Maintenance Faults 47
   RUNG wire#powerrail
      Contact( "BA040AZSCDR28_MendrelCathodeFrontAxisZ".StatusDrive.Error )
      { S7_Templates := "time_type := Time" } "Unit1.Em6.Alarms".tonMaintenanceFault[47].TON(pt := #DelayTime, et =>)
      wire#w1
      Move(in := "BA040AZSCDR28_MendrelCathodeFrontAxisZ".ErrorDetail.Number, out1 => "Unit1.Em6.Alarms".axisErrorCode[7])
   END_RUNG
   RUNG wire#w1
      S_Coil( "Unit1.Em6.Alarms".maintenanceFaults[47] )
   END_RUNG
   // the same network as SCL:
   "Unit1.Em6.Alarms".tonMaintenanceFault[47].TON(IN := "BA040AZSCDR28_MendrelCathodeFrontAxisZ".StatusDrive.Error,
                           PT := #DelayTime);
   IF "Unit1.Em6.Alarms".tonMaintenanceFault[47].Q THEN
       "Unit1.Em6.Alarms".axisErrorCode[7] := "BA040AZSCDR28_MendrelCathodeFrontAxisZ".ErrorDetail.Number;
       "Unit1.Em6.Alarms".maintenanceFaults[47] := TRUE;
   END_IF;
END_REGION

REGION Network 48: PFE Maintenance Faults 48
   RUNG wire#powerrail
      Contact( "BA040AZSCDR29_MendrelCathodeRearAxisY".StatusDrive.Error )
      { S7_Templates := "time_type := Time" } "Unit1.Em6.Alarms".tonMaintenanceFault[48].TON(pt := #DelayTime, et =>)
      wire#w1
      Move(in := "BA040AZSCDR29_MendrelCathodeRearAxisY".ErrorDetail.Number, out1 => "Unit1.Em6.Alarms".axisErrorCode[8])
   END_RUNG
   RUNG wire#w1
      S_Coil( "Unit1.Em6.Alarms".maintenanceFaults[48] )
   END_RUNG
   // the same network as SCL:
   "Unit1.Em6.Alarms".tonMaintenanceFault[48].TON(IN := "BA040AZSCDR29_MendrelCathodeRearAxisY".StatusDrive.Error,
                           PT := #DelayTime);
   IF "Unit1.Em6.Alarms".tonMaintenanceFault[48].Q THEN
       "Unit1.Em6.Alarms".axisErrorCode[8] := "BA040AZSCDR29_MendrelCathodeRearAxisY".ErrorDetail.Number;
       "Unit1.Em6.Alarms".maintenanceFaults[48] := TRUE;
   END_IF;
END_REGION

REGION Network 49: PFE Maintenance Faults 49
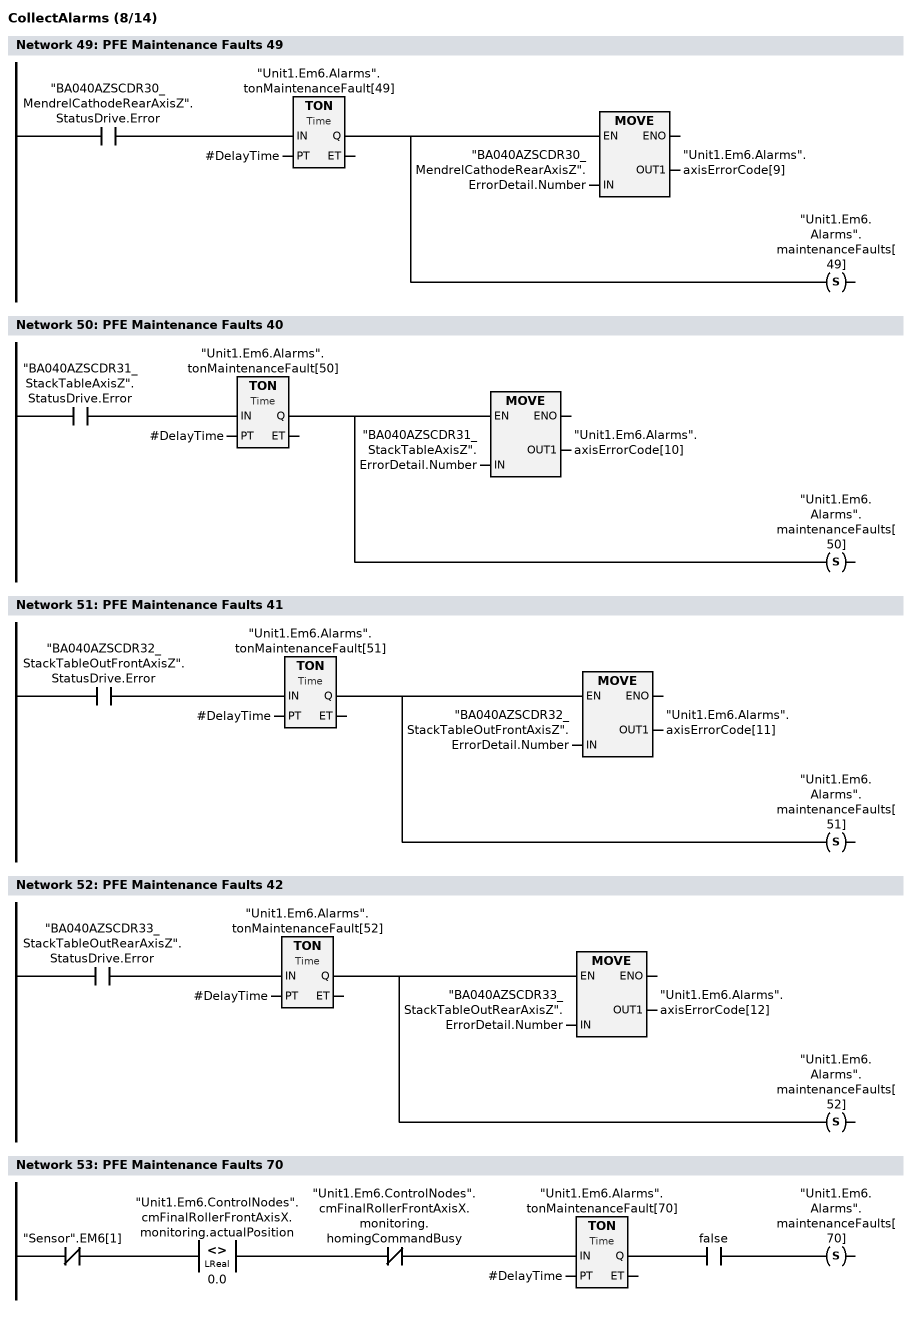
   RUNG wire#powerrail
      Contact( "BA040AZSCDR30_MendrelCathodeRearAxisZ".StatusDrive.Error )
      { S7_Templates := "time_type := Time" } "Unit1.Em6.Alarms".tonMaintenanceFault[49].TON(pt := #DelayTime, et =>)
      wire#w1
      Move(in := "BA040AZSCDR30_MendrelCathodeRearAxisZ".ErrorDetail.Number, out1 => "Unit1.Em6.Alarms".axisErrorCode[9])
   END_RUNG
   RUNG wire#w1
      S_Coil( "Unit1.Em6.Alarms".maintenanceFaults[49] )
   END_RUNG
   // the same network as SCL:
   "Unit1.Em6.Alarms".tonMaintenanceFault[49].TON(IN := "BA040AZSCDR30_MendrelCathodeRearAxisZ".StatusDrive.Error,
                           PT := #DelayTime);
   IF "Unit1.Em6.Alarms".tonMaintenanceFault[49].Q THEN
       "Unit1.Em6.Alarms".axisErrorCode[9] := "BA040AZSCDR30_MendrelCathodeRearAxisZ".ErrorDetail.Number;
       "Unit1.Em6.Alarms".maintenanceFaults[49] := TRUE;
   END_IF;
END_REGION

REGION Network 50: PFE Maintenance Faults 40
   RUNG wire#powerrail
      Contact( "BA040AZSCDR31_StackTableAxisZ".StatusDrive.Error )
      { S7_Templates := "time_type := Time" } "Unit1.Em6.Alarms".tonMaintenanceFault[50].TON(pt := #DelayTime, et =>)
      wire#w1
      Move(in := "BA040AZSCDR31_StackTableAxisZ".ErrorDetail.Number, out1 => "Unit1.Em6.Alarms".axisErrorCode[10])
   END_RUNG
   RUNG wire#w1
      S_Coil( "Unit1.Em6.Alarms".maintenanceFaults[50] )
   END_RUNG
   // the same network as SCL:
   "Unit1.Em6.Alarms".tonMaintenanceFault[50].TON(IN := "BA040AZSCDR31_StackTableAxisZ".StatusDrive.Error,
                           PT := #DelayTime);
   IF "Unit1.Em6.Alarms".tonMaintenanceFault[50].Q THEN
       "Unit1.Em6.Alarms".axisErrorCode[10] := "BA040AZSCDR31_StackTableAxisZ".ErrorDetail.Number;
       "Unit1.Em6.Alarms".maintenanceFaults[50] := TRUE;
   END_IF;
END_REGION

REGION Network 51: PFE Maintenance Faults 41
   RUNG wire#powerrail
      Contact( "BA040AZSCDR32_StackTableOutFrontAxisZ".StatusDrive.Error )
      { S7_Templates := "time_type := Time" } "Unit1.Em6.Alarms".tonMaintenanceFault[51].TON(pt := #DelayTime, et =>)
      wire#w1
      Move(in := "BA040AZSCDR32_StackTableOutFrontAxisZ".ErrorDetail.Number, out1 => "Unit1.Em6.Alarms".axisErrorCode[11])
   END_RUNG
   RUNG wire#w1
      S_Coil( "Unit1.Em6.Alarms".maintenanceFaults[51] )
   END_RUNG
   // the same network as SCL:
   "Unit1.Em6.Alarms".tonMaintenanceFault[51].TON(IN := "BA040AZSCDR32_StackTableOutFrontAxisZ".StatusDrive.Error,
                           PT := #DelayTime);
   IF "Unit1.Em6.Alarms".tonMaintenanceFault[51].Q THEN
       "Unit1.Em6.Alarms".axisErrorCode[11] := "BA040AZSCDR32_StackTableOutFrontAxisZ".ErrorDetail.Number;
       "Unit1.Em6.Alarms".maintenanceFaults[51] := TRUE;
   END_IF;
END_REGION

REGION Network 52: PFE Maintenance Faults 42
   RUNG wire#powerrail
      Contact( "BA040AZSCDR33_StackTableOutRearAxisZ".StatusDrive.Error )
      { S7_Templates := "time_type := Time" } "Unit1.Em6.Alarms".tonMaintenanceFault[52].TON(pt := #DelayTime, et =>)
      wire#w1
      Move(in := "BA040AZSCDR33_StackTableOutRearAxisZ".ErrorDetail.Number, out1 => "Unit1.Em6.Alarms".axisErrorCode[12])
   END_RUNG
   RUNG wire#w1
      S_Coil( "Unit1.Em6.Alarms".maintenanceFaults[52] )
   END_RUNG
   // the same network as SCL:
   "Unit1.Em6.Alarms".tonMaintenanceFault[52].TON(IN := "BA040AZSCDR33_StackTableOutRearAxisZ".StatusDrive.Error,
                           PT := #DelayTime);
   IF "Unit1.Em6.Alarms".tonMaintenanceFault[52].Q THEN
       "Unit1.Em6.Alarms".axisErrorCode[12] := "BA040AZSCDR33_StackTableOutRearAxisZ".ErrorDetail.Number;
       "Unit1.Em6.Alarms".maintenanceFaults[52] := TRUE;
   END_IF;
END_REGION

REGION Network 53: PFE Maintenance Faults 70
   RUNG wire#powerrail
      I_Contact( "Sensor".EM6[1] )
      { S7_Templates := "SrcType := LReal" } NE_Contact(in1 := "Unit1.Em6.ControlNodes".cmFinalRollerFrontAxisX.monitoring.actualPosition, in2 := 0.0)
      I_Contact( "Unit1.Em6.ControlNodes".cmFinalRollerFrontAxisX.monitoring.homingCommandBusy )
      { S7_Templates := "time_type := Time" } "Unit1.Em6.Alarms".tonMaintenanceFault[70].TON(pt := #DelayTime, et =>)
      Contact( false )
      S_Coil( "Unit1.Em6.Alarms".maintenanceFaults[70] )
   END_RUNG
   // the same network as SCL:
   "Unit1.Em6.Alarms".tonMaintenanceFault[70].TON(IN := NOT "Sensor".EM6[1] AND ("Unit1.Em6.ControlNodes".cmFinalRollerFrontAxisX.monitoring.actualPosition <> 0.0) AND NOT "Unit1.Em6.ControlNodes".cmFinalRollerFrontAxisX.monitoring.homingCommandBusy,
                           PT := #DelayTime);
   IF "Unit1.Em6.Alarms".tonMaintenanceFault[70].Q AND false THEN
       "Unit1.Em6.Alarms".maintenanceFaults[70] := TRUE;
   END_IF;
END_REGION

REGION Network 54: PFE Maintenance Faults 71
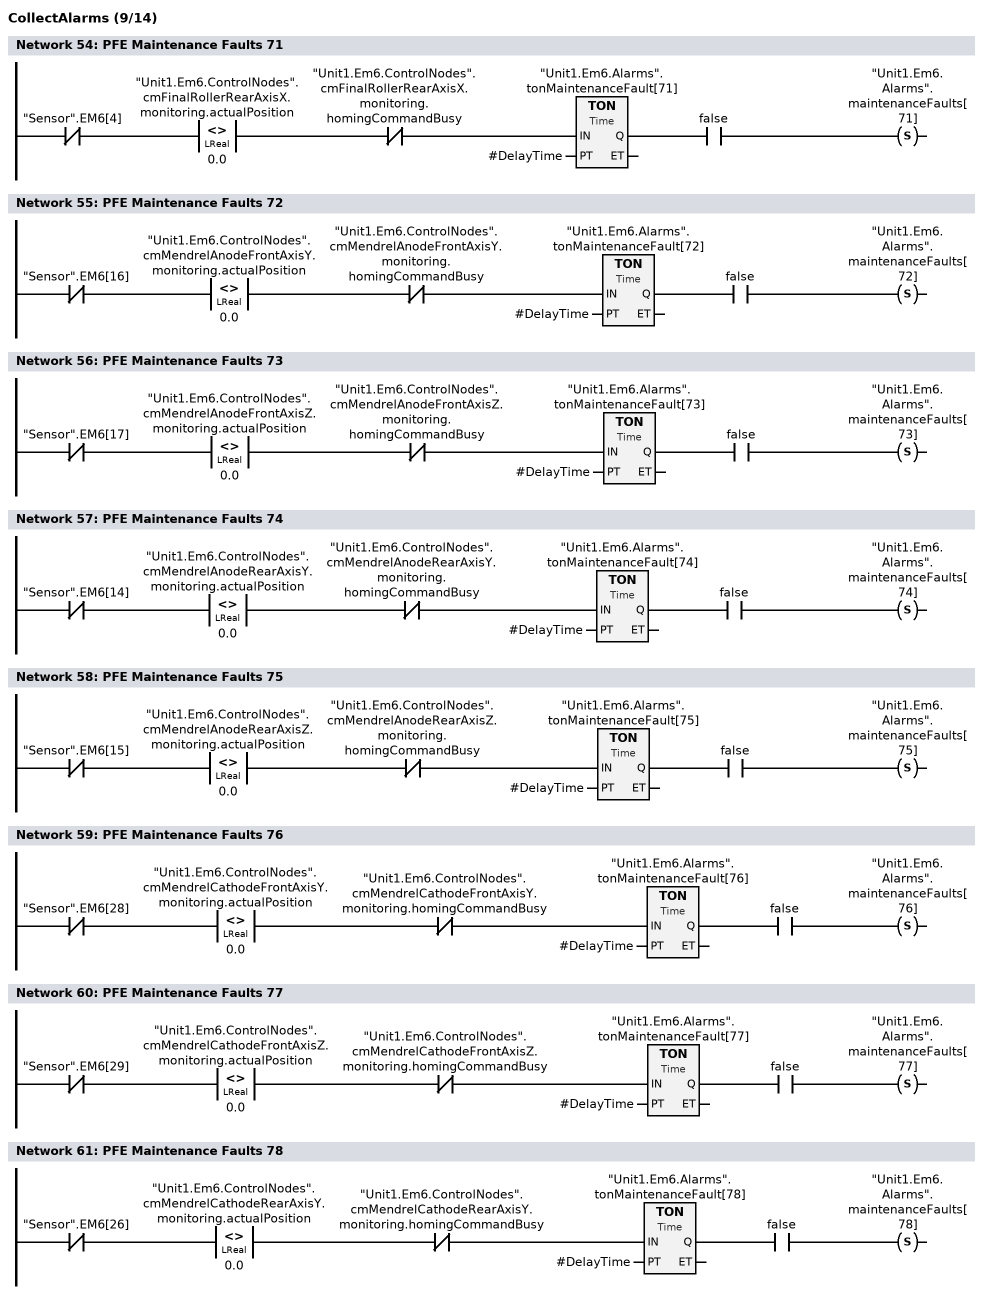
   RUNG wire#powerrail
      I_Contact( "Sensor".EM6[4] )
      { S7_Templates := "SrcType := LReal" } NE_Contact(in1 := "Unit1.Em6.ControlNodes".cmFinalRollerRearAxisX.monitoring.actualPosition, in2 := 0.0)
      I_Contact( "Unit1.Em6.ControlNodes".cmFinalRollerRearAxisX.monitoring.homingCommandBusy )
      { S7_Templates := "time_type := Time" } "Unit1.Em6.Alarms".tonMaintenanceFault[71].TON(pt := #DelayTime, et =>)
      Contact( false )
      S_Coil( "Unit1.Em6.Alarms".maintenanceFaults[71] )
   END_RUNG
   // the same network as SCL:
   "Unit1.Em6.Alarms".tonMaintenanceFault[71].TON(IN := NOT "Sensor".EM6[4] AND ("Unit1.Em6.ControlNodes".cmFinalRollerRearAxisX.monitoring.actualPosition <> 0.0) AND NOT "Unit1.Em6.ControlNodes".cmFinalRollerRearAxisX.monitoring.homingCommandBusy,
                           PT := #DelayTime);
   IF "Unit1.Em6.Alarms".tonMaintenanceFault[71].Q AND false THEN
       "Unit1.Em6.Alarms".maintenanceFaults[71] := TRUE;
   END_IF;
END_REGION

REGION Network 55: PFE Maintenance Faults 72
   RUNG wire#powerrail
      I_Contact( "Sensor".EM6[16] )
      { S7_Templates := "SrcType := LReal" } NE_Contact(in1 := "Unit1.Em6.ControlNodes".cmMendrelAnodeFrontAxisY.monitoring.actualPosition, in2 := 0.0)
      I_Contact( "Unit1.Em6.ControlNodes".cmMendrelAnodeFrontAxisY.monitoring.homingCommandBusy )
      { S7_Templates := "time_type := Time" } "Unit1.Em6.Alarms".tonMaintenanceFault[72].TON(pt := #DelayTime, et =>)
      Contact( false )
      S_Coil( "Unit1.Em6.Alarms".maintenanceFaults[72] )
   END_RUNG
   // the same network as SCL:
   "Unit1.Em6.Alarms".tonMaintenanceFault[72].TON(IN := NOT "Sensor".EM6[16] AND ("Unit1.Em6.ControlNodes".cmMendrelAnodeFrontAxisY.monitoring.actualPosition <> 0.0) AND NOT "Unit1.Em6.ControlNodes".cmMendrelAnodeFrontAxisY.monitoring.homingCommandBusy,
                           PT := #DelayTime);
   IF "Unit1.Em6.Alarms".tonMaintenanceFault[72].Q AND false THEN
       "Unit1.Em6.Alarms".maintenanceFaults[72] := TRUE;
   END_IF;
END_REGION

REGION Network 56: PFE Maintenance Faults 73
   RUNG wire#powerrail
      I_Contact( "Sensor".EM6[17] )
      { S7_Templates := "SrcType := LReal" } NE_Contact(in1 := "Unit1.Em6.ControlNodes".cmMendrelAnodeFrontAxisZ.monitoring.actualPosition, in2 := 0.0)
      I_Contact( "Unit1.Em6.ControlNodes".cmMendrelAnodeFrontAxisZ.monitoring.homingCommandBusy )
      { S7_Templates := "time_type := Time" } "Unit1.Em6.Alarms".tonMaintenanceFault[73].TON(pt := #DelayTime, et =>)
      Contact( false )
      S_Coil( "Unit1.Em6.Alarms".maintenanceFaults[73] )
   END_RUNG
   // the same network as SCL:
   "Unit1.Em6.Alarms".tonMaintenanceFault[73].TON(IN := NOT "Sensor".EM6[17] AND ("Unit1.Em6.ControlNodes".cmMendrelAnodeFrontAxisZ.monitoring.actualPosition <> 0.0) AND NOT "Unit1.Em6.ControlNodes".cmMendrelAnodeFrontAxisZ.monitoring.homingCommandBusy,
                           PT := #DelayTime);
   IF "Unit1.Em6.Alarms".tonMaintenanceFault[73].Q AND false THEN
       "Unit1.Em6.Alarms".maintenanceFaults[73] := TRUE;
   END_IF;
END_REGION

REGION Network 57: PFE Maintenance Faults 74
   RUNG wire#powerrail
      I_Contact( "Sensor".EM6[14] )
      { S7_Templates := "SrcType := LReal" } NE_Contact(in1 := "Unit1.Em6.ControlNodes".cmMendrelAnodeRearAxisY.monitoring.actualPosition, in2 := 0.0)
      I_Contact( "Unit1.Em6.ControlNodes".cmMendrelAnodeRearAxisY.monitoring.homingCommandBusy )
      { S7_Templates := "time_type := Time" } "Unit1.Em6.Alarms".tonMaintenanceFault[74].TON(pt := #DelayTime, et =>)
      Contact( false )
      S_Coil( "Unit1.Em6.Alarms".maintenanceFaults[74] )
   END_RUNG
   // the same network as SCL:
   "Unit1.Em6.Alarms".tonMaintenanceFault[74].TON(IN := NOT "Sensor".EM6[14] AND ("Unit1.Em6.ControlNodes".cmMendrelAnodeRearAxisY.monitoring.actualPosition <> 0.0) AND NOT "Unit1.Em6.ControlNodes".cmMendrelAnodeRearAxisY.monitoring.homingCommandBusy,
                           PT := #DelayTime);
   IF "Unit1.Em6.Alarms".tonMaintenanceFault[74].Q AND false THEN
       "Unit1.Em6.Alarms".maintenanceFaults[74] := TRUE;
   END_IF;
END_REGION

REGION Network 58: PFE Maintenance Faults 75
   RUNG wire#powerrail
      I_Contact( "Sensor".EM6[15] )
      { S7_Templates := "SrcType := LReal" } NE_Contact(in1 := "Unit1.Em6.ControlNodes".cmMendrelAnodeRearAxisZ.monitoring.actualPosition, in2 := 0.0)
      I_Contact( "Unit1.Em6.ControlNodes".cmMendrelAnodeRearAxisZ.monitoring.homingCommandBusy )
      { S7_Templates := "time_type := Time" } "Unit1.Em6.Alarms".tonMaintenanceFault[75].TON(pt := #DelayTime, et =>)
      Contact( false )
      S_Coil( "Unit1.Em6.Alarms".maintenanceFaults[75] )
   END_RUNG
   // the same network as SCL:
   "Unit1.Em6.Alarms".tonMaintenanceFault[75].TON(IN := NOT "Sensor".EM6[15] AND ("Unit1.Em6.ControlNodes".cmMendrelAnodeRearAxisZ.monitoring.actualPosition <> 0.0) AND NOT "Unit1.Em6.ControlNodes".cmMendrelAnodeRearAxisZ.monitoring.homingCommandBusy,
                           PT := #DelayTime);
   IF "Unit1.Em6.Alarms".tonMaintenanceFault[75].Q AND false THEN
       "Unit1.Em6.Alarms".maintenanceFaults[75] := TRUE;
   END_IF;
END_REGION

REGION Network 59: PFE Maintenance Faults 76
   RUNG wire#powerrail
      I_Contact( "Sensor".EM6[28] )
      { S7_Templates := "SrcType := LReal" } NE_Contact(in1 := "Unit1.Em6.ControlNodes".cmMendrelCathodeFrontAxisY.monitoring.actualPosition, in2 := 0.0)
      I_Contact( "Unit1.Em6.ControlNodes".cmMendrelCathodeFrontAxisY.monitoring.homingCommandBusy )
      { S7_Templates := "time_type := Time" } "Unit1.Em6.Alarms".tonMaintenanceFault[76].TON(pt := #DelayTime, et =>)
      Contact( false )
      S_Coil( "Unit1.Em6.Alarms".maintenanceFaults[76] )
   END_RUNG
   // the same network as SCL:
   "Unit1.Em6.Alarms".tonMaintenanceFault[76].TON(IN := NOT "Sensor".EM6[28] AND ("Unit1.Em6.ControlNodes".cmMendrelCathodeFrontAxisY.monitoring.actualPosition <> 0.0) AND NOT "Unit1.Em6.ControlNodes".cmMendrelCathodeFrontAxisY.monitoring.homingCommandBusy,
                           PT := #DelayTime);
   IF "Unit1.Em6.Alarms".tonMaintenanceFault[76].Q AND false THEN
       "Unit1.Em6.Alarms".maintenanceFaults[76] := TRUE;
   END_IF;
END_REGION

REGION Network 60: PFE Maintenance Faults 77
   RUNG wire#powerrail
      I_Contact( "Sensor".EM6[29] )
      { S7_Templates := "SrcType := LReal" } NE_Contact(in1 := "Unit1.Em6.ControlNodes".cmMendrelCathodeFrontAxisZ.monitoring.actualPosition, in2 := 0.0)
      I_Contact( "Unit1.Em6.ControlNodes".cmMendrelCathodeFrontAxisZ.monitoring.homingCommandBusy )
      { S7_Templates := "time_type := Time" } "Unit1.Em6.Alarms".tonMaintenanceFault[77].TON(pt := #DelayTime, et =>)
      Contact( false )
      S_Coil( "Unit1.Em6.Alarms".maintenanceFaults[77] )
   END_RUNG
   // the same network as SCL:
   "Unit1.Em6.Alarms".tonMaintenanceFault[77].TON(IN := NOT "Sensor".EM6[29] AND ("Unit1.Em6.ControlNodes".cmMendrelCathodeFrontAxisZ.monitoring.actualPosition <> 0.0) AND NOT "Unit1.Em6.ControlNodes".cmMendrelCathodeFrontAxisZ.monitoring.homingCommandBusy,
                           PT := #DelayTime);
   IF "Unit1.Em6.Alarms".tonMaintenanceFault[77].Q AND false THEN
       "Unit1.Em6.Alarms".maintenanceFaults[77] := TRUE;
   END_IF;
END_REGION

REGION Network 61: PFE Maintenance Faults 78
   RUNG wire#powerrail
      I_Contact( "Sensor".EM6[26] )
      { S7_Templates := "SrcType := LReal" } NE_Contact(in1 := "Unit1.Em6.ControlNodes".cmMendrelCathodeRearAxisY.monitoring.actualPosition, in2 := 0.0)
      I_Contact( "Unit1.Em6.ControlNodes".cmMendrelCathodeRearAxisY.monitoring.homingCommandBusy )
      { S7_Templates := "time_type := Time" } "Unit1.Em6.Alarms".tonMaintenanceFault[78].TON(pt := #DelayTime, et =>)
      Contact( false )
      S_Coil( "Unit1.Em6.Alarms".maintenanceFaults[78] )
   END_RUNG
   // the same network as SCL:
   "Unit1.Em6.Alarms".tonMaintenanceFault[78].TON(IN := NOT "Sensor".EM6[26] AND ("Unit1.Em6.ControlNodes".cmMendrelCathodeRearAxisY.monitoring.actualPosition <> 0.0) AND NOT "Unit1.Em6.ControlNodes".cmMendrelCathodeRearAxisY.monitoring.homingCommandBusy,
                           PT := #DelayTime);
   IF "Unit1.Em6.Alarms".tonMaintenanceFault[78].Q AND false THEN
       "Unit1.Em6.Alarms".maintenanceFaults[78] := TRUE;
   END_IF;
END_REGION

REGION Network 62: PFE Maintenance Faults 79
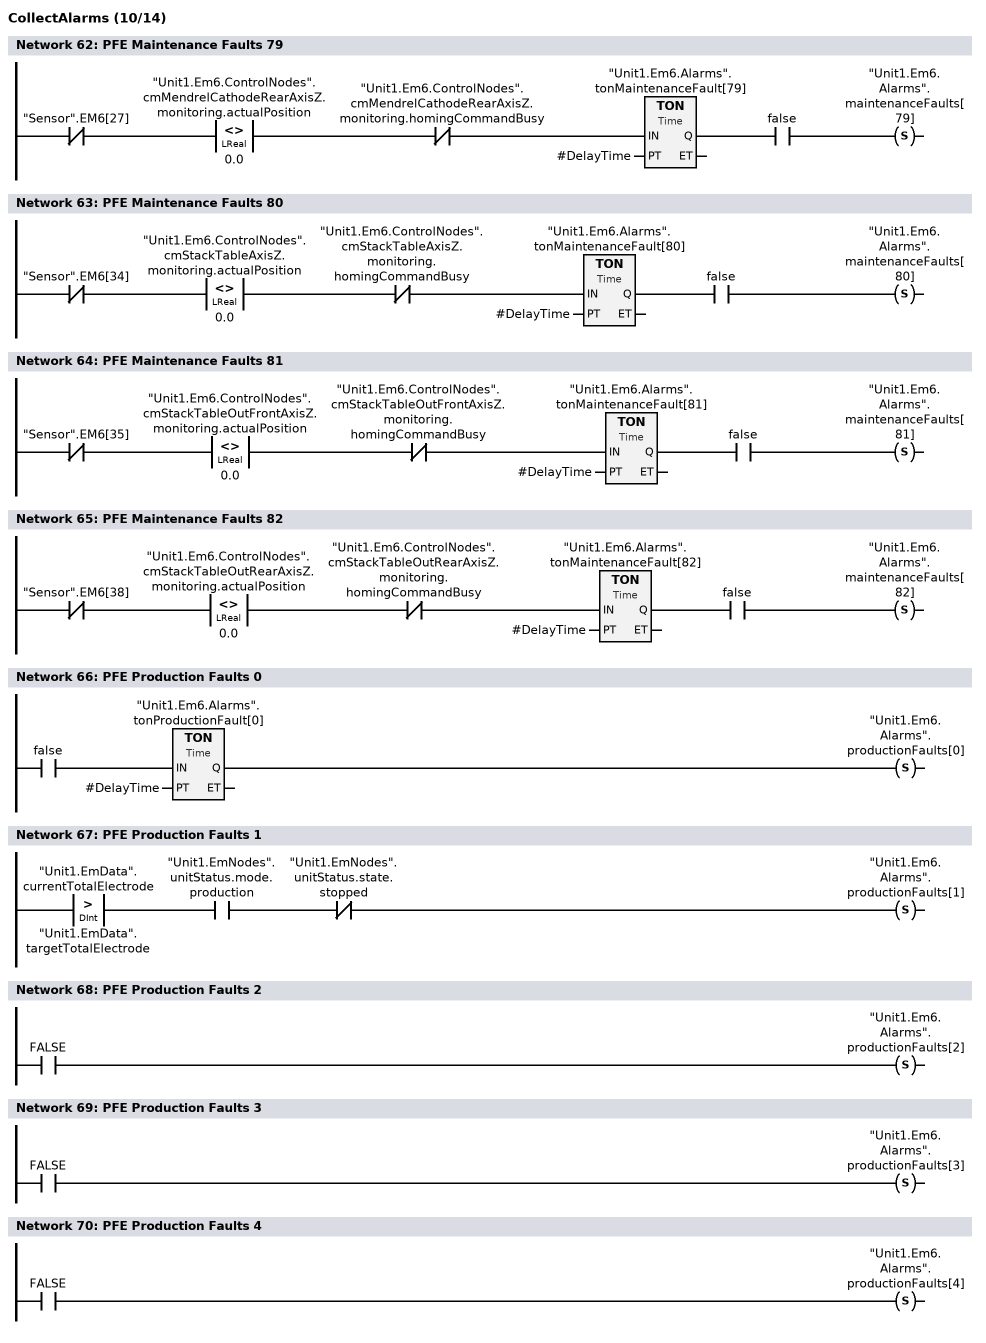
   RUNG wire#powerrail
      I_Contact( "Sensor".EM6[27] )
      { S7_Templates := "SrcType := LReal" } NE_Contact(in1 := "Unit1.Em6.ControlNodes".cmMendrelCathodeRearAxisZ.monitoring.actualPosition, in2 := 0.0)
      I_Contact( "Unit1.Em6.ControlNodes".cmMendrelCathodeRearAxisZ.monitoring.homingCommandBusy )
      { S7_Templates := "time_type := Time" } "Unit1.Em6.Alarms".tonMaintenanceFault[79].TON(pt := #DelayTime, et =>)
      Contact( false )
      S_Coil( "Unit1.Em6.Alarms".maintenanceFaults[79] )
   END_RUNG
   // the same network as SCL:
   "Unit1.Em6.Alarms".tonMaintenanceFault[79].TON(IN := NOT "Sensor".EM6[27] AND ("Unit1.Em6.ControlNodes".cmMendrelCathodeRearAxisZ.monitoring.actualPosition <> 0.0) AND NOT "Unit1.Em6.ControlNodes".cmMendrelCathodeRearAxisZ.monitoring.homingCommandBusy,
                           PT := #DelayTime);
   IF "Unit1.Em6.Alarms".tonMaintenanceFault[79].Q AND false THEN
       "Unit1.Em6.Alarms".maintenanceFaults[79] := TRUE;
   END_IF;
END_REGION

REGION Network 63: PFE Maintenance Faults 80
   RUNG wire#powerrail
      I_Contact( "Sensor".EM6[34] )
      { S7_Templates := "SrcType := LReal" } NE_Contact(in1 := "Unit1.Em6.ControlNodes".cmStackTableAxisZ.monitoring.actualPosition, in2 := 0.0)
      I_Contact( "Unit1.Em6.ControlNodes".cmStackTableAxisZ.monitoring.homingCommandBusy )
      { S7_Templates := "time_type := Time" } "Unit1.Em6.Alarms".tonMaintenanceFault[80].TON(pt := #DelayTime, et =>)
      Contact( false )
      S_Coil( "Unit1.Em6.Alarms".maintenanceFaults[80] )
   END_RUNG
   // the same network as SCL:
   "Unit1.Em6.Alarms".tonMaintenanceFault[80].TON(IN := NOT "Sensor".EM6[34] AND ("Unit1.Em6.ControlNodes".cmStackTableAxisZ.monitoring.actualPosition <> 0.0) AND NOT "Unit1.Em6.ControlNodes".cmStackTableAxisZ.monitoring.homingCommandBusy,
                           PT := #DelayTime);
   IF "Unit1.Em6.Alarms".tonMaintenanceFault[80].Q AND false THEN
       "Unit1.Em6.Alarms".maintenanceFaults[80] := TRUE;
   END_IF;
END_REGION

REGION Network 64: PFE Maintenance Faults 81
   RUNG wire#powerrail
      I_Contact( "Sensor".EM6[35] )
      { S7_Templates := "SrcType := LReal" } NE_Contact(in1 := "Unit1.Em6.ControlNodes".cmStackTableOutFrontAxisZ.monitoring.actualPosition, in2 := 0.0)
      I_Contact( "Unit1.Em6.ControlNodes".cmStackTableOutFrontAxisZ.monitoring.homingCommandBusy )
      { S7_Templates := "time_type := Time" } "Unit1.Em6.Alarms".tonMaintenanceFault[81].TON(pt := #DelayTime, et =>)
      Contact( false )
      S_Coil( "Unit1.Em6.Alarms".maintenanceFaults[81] )
   END_RUNG
   // the same network as SCL:
   "Unit1.Em6.Alarms".tonMaintenanceFault[81].TON(IN := NOT "Sensor".EM6[35] AND ("Unit1.Em6.ControlNodes".cmStackTableOutFrontAxisZ.monitoring.actualPosition <> 0.0) AND NOT "Unit1.Em6.ControlNodes".cmStackTableOutFrontAxisZ.monitoring.homingCommandBusy,
                           PT := #DelayTime);
   IF "Unit1.Em6.Alarms".tonMaintenanceFault[81].Q AND false THEN
       "Unit1.Em6.Alarms".maintenanceFaults[81] := TRUE;
   END_IF;
END_REGION

REGION Network 65: PFE Maintenance Faults 82
   RUNG wire#powerrail
      I_Contact( "Sensor".EM6[38] )
      { S7_Templates := "SrcType := LReal" } NE_Contact(in1 := "Unit1.Em6.ControlNodes".cmStackTableOutRearAxisZ.monitoring.actualPosition, in2 := 0.0)
      I_Contact( "Unit1.Em6.ControlNodes".cmStackTableOutRearAxisZ.monitoring.homingCommandBusy )
      { S7_Templates := "time_type := Time" } "Unit1.Em6.Alarms".tonMaintenanceFault[82].TON(pt := #DelayTime, et =>)
      Contact( false )
      S_Coil( "Unit1.Em6.Alarms".maintenanceFaults[82] )
   END_RUNG
   // the same network as SCL:
   "Unit1.Em6.Alarms".tonMaintenanceFault[82].TON(IN := NOT "Sensor".EM6[38] AND ("Unit1.Em6.ControlNodes".cmStackTableOutRearAxisZ.monitoring.actualPosition <> 0.0) AND NOT "Unit1.Em6.ControlNodes".cmStackTableOutRearAxisZ.monitoring.homingCommandBusy,
                           PT := #DelayTime);
   IF "Unit1.Em6.Alarms".tonMaintenanceFault[82].Q AND false THEN
       "Unit1.Em6.Alarms".maintenanceFaults[82] := TRUE;
   END_IF;
END_REGION

REGION Network 66: PFE Production Faults 0
   RUNG wire#powerrail
      Contact( false )
      { S7_Templates := "time_type := Time" } "Unit1.Em6.Alarms".tonProductionFault[0].TON(pt := #DelayTime, et =>)
      S_Coil( "Unit1.Em6.Alarms".productionFaults[0] )
   END_RUNG
   // the same network as SCL:
   "Unit1.Em6.Alarms".tonProductionFault[0].TON(IN := false, PT := #DelayTime);
   IF "Unit1.Em6.Alarms".tonProductionFault[0].Q THEN "Unit1.Em6.Alarms".productionFaults[0] := TRUE; END_IF;
END_REGION

REGION Network 67: PFE Production Faults 1
   RUNG wire#powerrail
      { S7_Templates := "SrcType := DInt" } GT_Contact(in1 := "Unit1.EmData".currentTotalElectrode, in2 := "Unit1.EmData".targetTotalElectrode)
      Contact( "Unit1.EmNodes".unitStatus.mode.production )
      I_Contact( "Unit1.EmNodes".unitStatus.state.stopped )
      S_Coil( "Unit1.Em6.Alarms".productionFaults[1] )
   END_RUNG
   // the same network as SCL:
   IF ("Unit1.EmData".currentTotalElectrode > "Unit1.EmData".targetTotalElectrode) AND "Unit1.EmNodes".unitStatus.mode.production AND NOT "Unit1.EmNodes".unitStatus.state.stopped THEN
       "Unit1.Em6.Alarms".productionFaults[1] := TRUE;
   END_IF;
END_REGION

REGION Network 68: PFE Production Faults 2
   RUNG wire#powerrail
      Contact( FALSE )
      S_Coil( "Unit1.Em6.Alarms".productionFaults[2] )
   END_RUNG
   // the same network as SCL:
   IF FALSE THEN "Unit1.Em6.Alarms".productionFaults[2] := TRUE; END_IF;
END_REGION

REGION Network 69: PFE Production Faults 3
   RUNG wire#powerrail
      Contact( FALSE )
      S_Coil( "Unit1.Em6.Alarms".productionFaults[3] )
   END_RUNG
   // the same network as SCL:
   IF FALSE THEN "Unit1.Em6.Alarms".productionFaults[3] := TRUE; END_IF;
END_REGION

REGION Network 70: PFE Production Faults 4
   RUNG wire#powerrail
      Contact( FALSE )
      S_Coil( "Unit1.Em6.Alarms".productionFaults[4] )
   END_RUNG
   // the same network as SCL:
   IF FALSE THEN "Unit1.Em6.Alarms".productionFaults[4] := TRUE; END_IF;
END_REGION

REGION Network 71: PFE Tooling Faults 0
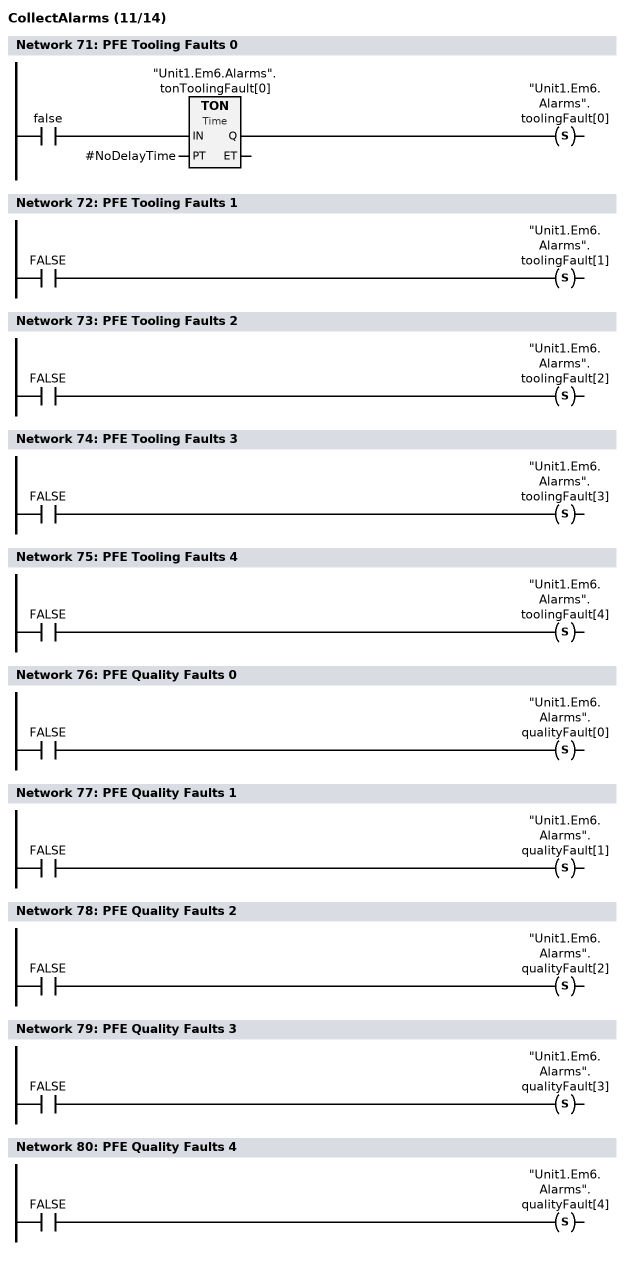
   RUNG wire#powerrail
      Contact( false )
      { S7_Templates := "time_type := Time" } "Unit1.Em6.Alarms".tonToolingFault[0].TON(pt := #NoDelayTime, et =>)
      S_Coil( "Unit1.Em6.Alarms".toolingFault[0] )
   END_RUNG
   // the same network as SCL:
   "Unit1.Em6.Alarms".tonToolingFault[0].TON(IN := false, PT := #NoDelayTime);
   IF "Unit1.Em6.Alarms".tonToolingFault[0].Q THEN "Unit1.Em6.Alarms".toolingFault[0] := TRUE; END_IF;
END_REGION

REGION Network 72: PFE Tooling Faults 1
   RUNG wire#powerrail
      Contact( FALSE )
      S_Coil( "Unit1.Em6.Alarms".toolingFault[1] )
   END_RUNG
   // the same network as SCL:
   IF FALSE THEN "Unit1.Em6.Alarms".toolingFault[1] := TRUE; END_IF;
END_REGION

REGION Network 73: PFE Tooling Faults 2
   RUNG wire#powerrail
      Contact( FALSE )
      S_Coil( "Unit1.Em6.Alarms".toolingFault[2] )
   END_RUNG
   // the same network as SCL:
   IF FALSE THEN "Unit1.Em6.Alarms".toolingFault[2] := TRUE; END_IF;
END_REGION

REGION Network 74: PFE Tooling Faults 3
   RUNG wire#powerrail
      Contact( FALSE )
      S_Coil( "Unit1.Em6.Alarms".toolingFault[3] )
   END_RUNG
   // the same network as SCL:
   IF FALSE THEN "Unit1.Em6.Alarms".toolingFault[3] := TRUE; END_IF;
END_REGION

REGION Network 75: PFE Tooling Faults 4
   RUNG wire#powerrail
      Contact( FALSE )
      S_Coil( "Unit1.Em6.Alarms".toolingFault[4] )
   END_RUNG
   // the same network as SCL:
   IF FALSE THEN "Unit1.Em6.Alarms".toolingFault[4] := TRUE; END_IF;
END_REGION

REGION Network 76: PFE Quality Faults 0
   RUNG wire#powerrail
      Contact( FALSE )
      S_Coil( "Unit1.Em6.Alarms".qualityFault[0] )
   END_RUNG
   // the same network as SCL:
   IF FALSE THEN "Unit1.Em6.Alarms".qualityFault[0] := TRUE; END_IF;
END_REGION

REGION Network 77: PFE Quality Faults 1
   RUNG wire#powerrail
      Contact( FALSE )
      S_Coil( "Unit1.Em6.Alarms".qualityFault[1] )
   END_RUNG
   // the same network as SCL:
   IF FALSE THEN "Unit1.Em6.Alarms".qualityFault[1] := TRUE; END_IF;
END_REGION

REGION Network 78: PFE Quality Faults 2
   RUNG wire#powerrail
      Contact( FALSE )
      S_Coil( "Unit1.Em6.Alarms".qualityFault[2] )
   END_RUNG
   // the same network as SCL:
   IF FALSE THEN "Unit1.Em6.Alarms".qualityFault[2] := TRUE; END_IF;
END_REGION

REGION Network 79: PFE Quality Faults 3
   RUNG wire#powerrail
      Contact( FALSE )
      S_Coil( "Unit1.Em6.Alarms".qualityFault[3] )
   END_RUNG
   // the same network as SCL:
   IF FALSE THEN "Unit1.Em6.Alarms".qualityFault[3] := TRUE; END_IF;
END_REGION

REGION Network 80: PFE Quality Faults 4
   RUNG wire#powerrail
      Contact( FALSE )
      S_Coil( "Unit1.Em6.Alarms".qualityFault[4] )
   END_RUNG
   // the same network as SCL:
   IF FALSE THEN "Unit1.Em6.Alarms".qualityFault[4] := TRUE; END_IF;
END_REGION

REGION Network 81: PFE Throughput Fault Blocked 0
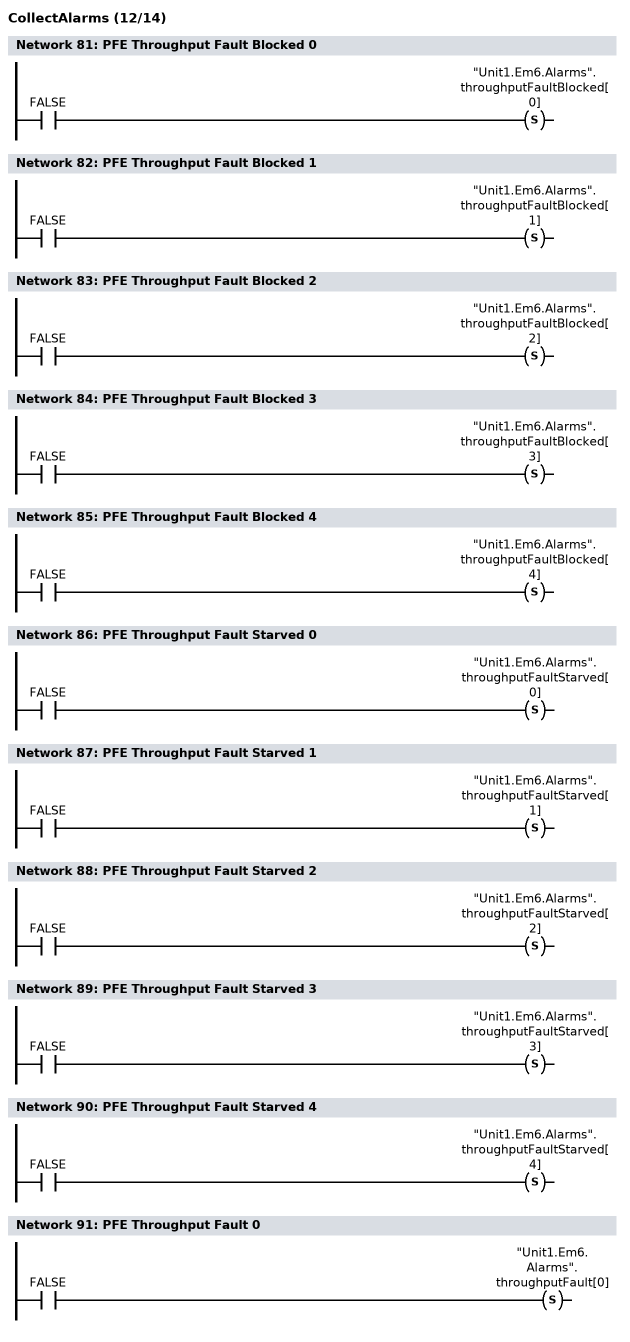
   RUNG wire#powerrail
      Contact( FALSE )
      S_Coil( "Unit1.Em6.Alarms".throughputFaultBlocked[0] )
   END_RUNG
   // the same network as SCL:
   IF FALSE THEN "Unit1.Em6.Alarms".throughputFaultBlocked[0] := TRUE; END_IF;
END_REGION

REGION Network 82: PFE Throughput Fault Blocked 1
   RUNG wire#powerrail
      Contact( FALSE )
      S_Coil( "Unit1.Em6.Alarms".throughputFaultBlocked[1] )
   END_RUNG
   // the same network as SCL:
   IF FALSE THEN "Unit1.Em6.Alarms".throughputFaultBlocked[1] := TRUE; END_IF;
END_REGION

REGION Network 83: PFE Throughput Fault Blocked 2
   RUNG wire#powerrail
      Contact( FALSE )
      S_Coil( "Unit1.Em6.Alarms".throughputFaultBlocked[2] )
   END_RUNG
   // the same network as SCL:
   IF FALSE THEN "Unit1.Em6.Alarms".throughputFaultBlocked[2] := TRUE; END_IF;
END_REGION

REGION Network 84: PFE Throughput Fault Blocked 3
   RUNG wire#powerrail
      Contact( FALSE )
      S_Coil( "Unit1.Em6.Alarms".throughputFaultBlocked[3] )
   END_RUNG
   // the same network as SCL:
   IF FALSE THEN "Unit1.Em6.Alarms".throughputFaultBlocked[3] := TRUE; END_IF;
END_REGION

REGION Network 85: PFE Throughput Fault Blocked 4
   RUNG wire#powerrail
      Contact( FALSE )
      S_Coil( "Unit1.Em6.Alarms".throughputFaultBlocked[4] )
   END_RUNG
   // the same network as SCL:
   IF FALSE THEN "Unit1.Em6.Alarms".throughputFaultBlocked[4] := TRUE; END_IF;
END_REGION

REGION Network 86: PFE Throughput Fault Starved 0
   RUNG wire#powerrail
      Contact( FALSE )
      S_Coil( "Unit1.Em6.Alarms".throughputFaultStarved[0] )
   END_RUNG
   // the same network as SCL:
   IF FALSE THEN "Unit1.Em6.Alarms".throughputFaultStarved[0] := TRUE; END_IF;
END_REGION

REGION Network 87: PFE Throughput Fault Starved 1
   RUNG wire#powerrail
      Contact( FALSE )
      S_Coil( "Unit1.Em6.Alarms".throughputFaultStarved[1] )
   END_RUNG
   // the same network as SCL:
   IF FALSE THEN "Unit1.Em6.Alarms".throughputFaultStarved[1] := TRUE; END_IF;
END_REGION

REGION Network 88: PFE Throughput Fault Starved 2
   RUNG wire#powerrail
      Contact( FALSE )
      S_Coil( "Unit1.Em6.Alarms".throughputFaultStarved[2] )
   END_RUNG
   // the same network as SCL:
   IF FALSE THEN "Unit1.Em6.Alarms".throughputFaultStarved[2] := TRUE; END_IF;
END_REGION

REGION Network 89: PFE Throughput Fault Starved 3
   RUNG wire#powerrail
      Contact( FALSE )
      S_Coil( "Unit1.Em6.Alarms".throughputFaultStarved[3] )
   END_RUNG
   // the same network as SCL:
   IF FALSE THEN "Unit1.Em6.Alarms".throughputFaultStarved[3] := TRUE; END_IF;
END_REGION

REGION Network 90: PFE Throughput Fault Starved 4
   RUNG wire#powerrail
      Contact( FALSE )
      S_Coil( "Unit1.Em6.Alarms".throughputFaultStarved[4] )
   END_RUNG
   // the same network as SCL:
   IF FALSE THEN "Unit1.Em6.Alarms".throughputFaultStarved[4] := TRUE; END_IF;
END_REGION

REGION Network 91: PFE Throughput Fault 0
   RUNG wire#powerrail
      Contact( FALSE )
      S_Coil( "Unit1.Em6.Alarms".throughputFault[0] )
   END_RUNG
   // the same network as SCL:
   IF FALSE THEN "Unit1.Em6.Alarms".throughputFault[0] := TRUE; END_IF;
END_REGION

REGION Network 92: PFE Throughput Fault 1
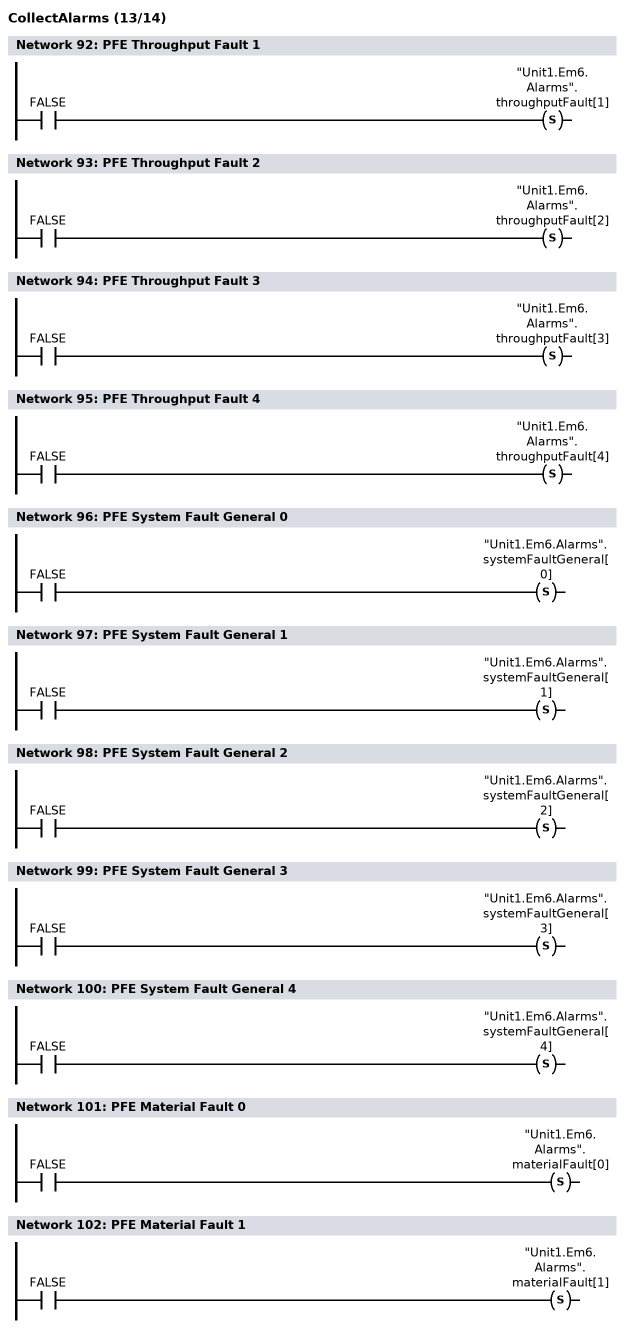
   RUNG wire#powerrail
      Contact( FALSE )
      S_Coil( "Unit1.Em6.Alarms".throughputFault[1] )
   END_RUNG
   // the same network as SCL:
   IF FALSE THEN "Unit1.Em6.Alarms".throughputFault[1] := TRUE; END_IF;
END_REGION

REGION Network 93: PFE Throughput Fault 2
   RUNG wire#powerrail
      Contact( FALSE )
      S_Coil( "Unit1.Em6.Alarms".throughputFault[2] )
   END_RUNG
   // the same network as SCL:
   IF FALSE THEN "Unit1.Em6.Alarms".throughputFault[2] := TRUE; END_IF;
END_REGION

REGION Network 94: PFE Throughput Fault 3
   RUNG wire#powerrail
      Contact( FALSE )
      S_Coil( "Unit1.Em6.Alarms".throughputFault[3] )
   END_RUNG
   // the same network as SCL:
   IF FALSE THEN "Unit1.Em6.Alarms".throughputFault[3] := TRUE; END_IF;
END_REGION

REGION Network 95: PFE Throughput Fault 4
   RUNG wire#powerrail
      Contact( FALSE )
      S_Coil( "Unit1.Em6.Alarms".throughputFault[4] )
   END_RUNG
   // the same network as SCL:
   IF FALSE THEN "Unit1.Em6.Alarms".throughputFault[4] := TRUE; END_IF;
END_REGION

REGION Network 96: PFE System Fault General 0
   RUNG wire#powerrail
      Contact( FALSE )
      S_Coil( "Unit1.Em6.Alarms".systemFaultGeneral[0] )
   END_RUNG
   // the same network as SCL:
   IF FALSE THEN "Unit1.Em6.Alarms".systemFaultGeneral[0] := TRUE; END_IF;
END_REGION

REGION Network 97: PFE System Fault General 1
   RUNG wire#powerrail
      Contact( FALSE )
      S_Coil( "Unit1.Em6.Alarms".systemFaultGeneral[1] )
   END_RUNG
   // the same network as SCL:
   IF FALSE THEN "Unit1.Em6.Alarms".systemFaultGeneral[1] := TRUE; END_IF;
END_REGION

REGION Network 98: PFE System Fault General 2
   RUNG wire#powerrail
      Contact( FALSE )
      S_Coil( "Unit1.Em6.Alarms".systemFaultGeneral[2] )
   END_RUNG
   // the same network as SCL:
   IF FALSE THEN "Unit1.Em6.Alarms".systemFaultGeneral[2] := TRUE; END_IF;
END_REGION

REGION Network 99: PFE System Fault General 3
   RUNG wire#powerrail
      Contact( FALSE )
      S_Coil( "Unit1.Em6.Alarms".systemFaultGeneral[3] )
   END_RUNG
   // the same network as SCL:
   IF FALSE THEN "Unit1.Em6.Alarms".systemFaultGeneral[3] := TRUE; END_IF;
END_REGION

REGION Network 100: PFE System Fault General 4
   RUNG wire#powerrail
      Contact( FALSE )
      S_Coil( "Unit1.Em6.Alarms".systemFaultGeneral[4] )
   END_RUNG
   // the same network as SCL:
   IF FALSE THEN "Unit1.Em6.Alarms".systemFaultGeneral[4] := TRUE; END_IF;
END_REGION

REGION Network 101: PFE Material Fault 0
   RUNG wire#powerrail
      Contact( FALSE )
      S_Coil( "Unit1.Em6.Alarms".materialFault[0] )
   END_RUNG
   // the same network as SCL:
   IF FALSE THEN "Unit1.Em6.Alarms".materialFault[0] := TRUE; END_IF;
END_REGION

REGION Network 102: PFE Material Fault 1
   RUNG wire#powerrail
      Contact( FALSE )
      S_Coil( "Unit1.Em6.Alarms".materialFault[1] )
   END_RUNG
   // the same network as SCL:
   IF FALSE THEN "Unit1.Em6.Alarms".materialFault[1] := TRUE; END_IF;
END_REGION

REGION Network 103: PFE Material Fault 2
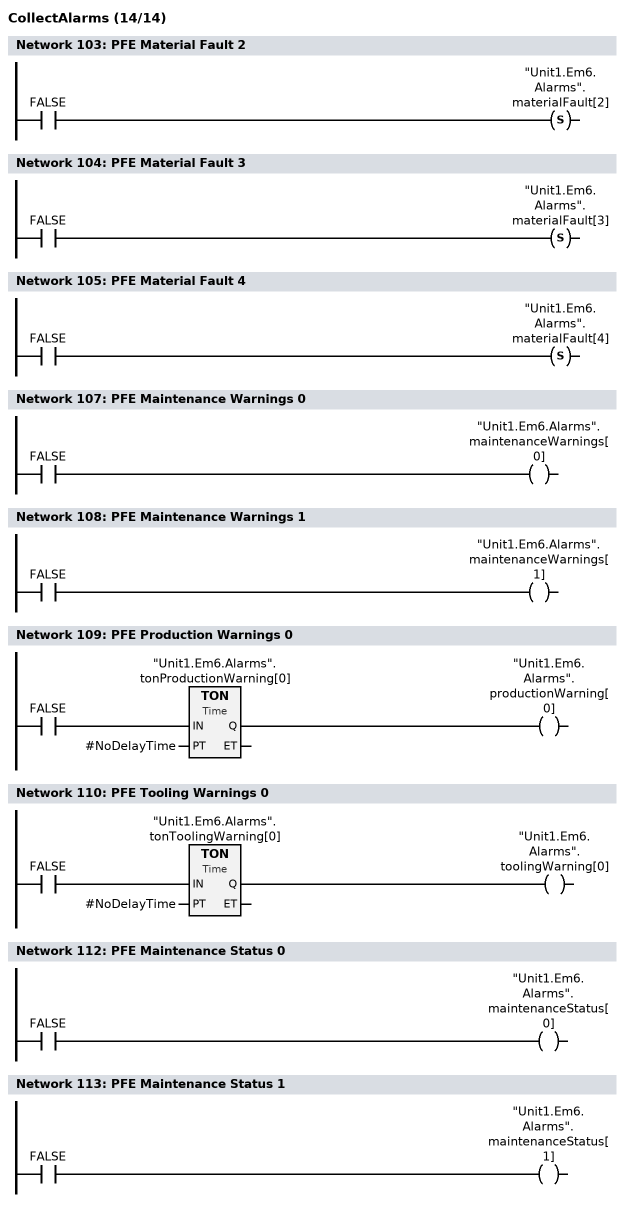
   RUNG wire#powerrail
      Contact( FALSE )
      S_Coil( "Unit1.Em6.Alarms".materialFault[2] )
   END_RUNG
   // the same network as SCL:
   IF FALSE THEN "Unit1.Em6.Alarms".materialFault[2] := TRUE; END_IF;
END_REGION

REGION Network 104: PFE Material Fault 3
   RUNG wire#powerrail
      Contact( FALSE )
      S_Coil( "Unit1.Em6.Alarms".materialFault[3] )
   END_RUNG
   // the same network as SCL:
   IF FALSE THEN "Unit1.Em6.Alarms".materialFault[3] := TRUE; END_IF;
END_REGION

REGION Network 105: PFE Material Fault 4
   RUNG wire#powerrail
      Contact( FALSE )
      S_Coil( "Unit1.Em6.Alarms".materialFault[4] )
   END_RUNG
   // the same network as SCL:
   IF FALSE THEN "Unit1.Em6.Alarms".materialFault[4] := TRUE; END_IF;
END_REGION

REGION Network 106: *************** Warning **************************
END_REGION

REGION Network 107: PFE Maintenance Warnings 0
   RUNG wire#powerrail
      Contact( FALSE )
      Coil( "Unit1.Em6.Alarms".maintenanceWarnings[0] )
   END_RUNG
   // the same network as SCL:
   "Unit1.Em6.Alarms".maintenanceWarnings[0] := FALSE;
END_REGION

REGION Network 108: PFE Maintenance Warnings 1
   RUNG wire#powerrail
      Contact( FALSE )
      Coil( "Unit1.Em6.Alarms".maintenanceWarnings[1] )
   END_RUNG
   // the same network as SCL:
   "Unit1.Em6.Alarms".maintenanceWarnings[1] := FALSE;
END_REGION

REGION Network 109: PFE Production Warnings 0
   RUNG wire#powerrail
      Contact( FALSE )
      { S7_Templates := "time_type := Time" } "Unit1.Em6.Alarms".tonProductionWarning[0].TON(pt := #NoDelayTime, et =>)
      Coil( "Unit1.Em6.Alarms".productionWarning[0] )
   END_RUNG
   // the same network as SCL:
   "Unit1.Em6.Alarms".tonProductionWarning[0].TON(IN := FALSE, PT := #NoDelayTime);
   "Unit1.Em6.Alarms".productionWarning[0] := "Unit1.Em6.Alarms".tonProductionWarning[0].Q;
END_REGION

REGION Network 110: PFE Tooling Warnings 0
   RUNG wire#powerrail
      Contact( FALSE )
      { S7_Templates := "time_type := Time" } "Unit1.Em6.Alarms".tonToolingWarning[0].TON(pt := #NoDelayTime, et =>)
      Coil( "Unit1.Em6.Alarms".toolingWarning[0] )
   END_RUNG
   // the same network as SCL:
   "Unit1.Em6.Alarms".tonToolingWarning[0].TON(IN := FALSE, PT := #NoDelayTime);
   "Unit1.Em6.Alarms".toolingWarning[0] := "Unit1.Em6.Alarms".tonToolingWarning[0].Q;
END_REGION

REGION Network 111: *************** Status ***************************
END_REGION

REGION Network 112: PFE Maintenance Status 0
   RUNG wire#powerrail
      Contact( FALSE )
      Coil( "Unit1.Em6.Alarms".maintenanceStatus[0] )
   END_RUNG
   // the same network as SCL:
   "Unit1.Em6.Alarms".maintenanceStatus[0] := FALSE;
END_REGION

REGION Network 113: PFE Maintenance Status 1
   RUNG wire#powerrail
      Contact( FALSE )
      Coil( "Unit1.Em6.Alarms".maintenanceStatus[1] )
   END_RUNG
   // the same network as SCL:
   "Unit1.Em6.Alarms".maintenanceStatus[1] := FALSE;
END_REGION
END_FUNCTION
